(* CODESYS project lateral_levitation_control_new.library
   TcLibraryId: TE140x Module Vendor|lateral_levitation_control_new|0.0.0.4
   Company: TE140x Module Vendor
   Title: lateral_levitation_control_new
   Placeholder: lateral_levitation_control_new
   Version: 0.0.0.4

Project tree, tasks and I/O mapping:
  POUs/
    function block FB_lateral_levitation_control_new [ST]: FB_exit, FB_init, nHResult, eInitExceptionHandling, eUpdateExceptionHandling, nExceptionCnt, stActiveException, bInitialized, bExecute
    TcCOM Wrapper/
      function block FB_lateral_levitation_control_new_TcCOM_InitStruct [ST]: FB_init, FB_afterinit, Reinit, FB_exit, eObjectState, nHResult, ipTcComObject, ipADI, nTaskOid, nTaskPriority, nTaskCycleTimeNs, nTaskPort, nTaskSortOrder, eTraceLevelMax, eModuleCaller, eCallerVerification, eStepSizeAdaptation, eExecutionSequence, bExecute, eAccessLockState, eInitExceptionHandling, eUpdateExceptionHandling, stModuleBuildInfo, bInitialized, nSkippedExecutionCount, stLibraryInfo, stModuleInfo, stModuleGeneratorInfo, stSimulinkModelInfo, elateral_levitation_control_new_P_Sharing, nlateral_levitation_control_new_P_Definer, stlateral_levitation_control_new_P, fSimulationTime, nCycleCount, nExceptionCount, stExceptionInfo
  DUTs/
    data type ST_FB_lateral_levitation_control_new_FB_Main
    data type ST_FB_lateral_levitation_control_new_FB_exit
    data type ST_FB_lateral_levitation_control_new_FB_init
    data type ST_GetSet_HRESULT
    data type E_FpExcptCtrlSetEx
    data type ST_GetSet_E_FpExcptCtrlSetEx
    data type ST_GetSet_ULINT
    data type ST_ExceptionInfo
    data type ST_GetSet_ST_ExceptionInfo
    data type ST_GetSet_BOOL
    data type T_matrix2xdouble
    data type T_matrix4xdouble
    data type E_SimTimeStep
    data type E_SolverMode
    data type E_ssMatrixType
    data type ST_RTWRTModelMethodsInfo
    data type E_slJmBdControl
    data type ST_ssSolverInfo
    data type T_matrix3xdouble
    data type T_matrix4xlogical
    data type ST_B_MATLABFunction2_lateral_levitation_control_new_T
    data type ST_B_lateral_levitation_control_new_T
    data type T_ZCSigState
    data type T_matrix2xZCSigState
    data type ST_PrevZCX_lateral_levitation_control_new_T
    data type ST_X_lateral_levitation_control_new_T
    data type ST_ExtU_lateral_levitation_control_new_T
    data type ST_ExtY_lateral_levitation_control_new_T
    data type T_matrix2xbool
    data type ST_XDis_lateral_levitation_control_new_T
    data type T_matrix8xdouble
    data type T_matrix8x4xdouble
    data type PLREAL
    data type T_matrix4xdoublepointer
    data type ST_ODE4_IntgData
    data type ST_DW_lateral_levitation_control_new_T
    data type ST_x08a7a7bbd0e5d629f7d70ceec84eacfe
    data type ST_xf09845edab6c83520d8d57def6d6fe1c
    data type ST_RT_MODEL_lateral_levitation_control_new_T
    data type T_matrix14xdouble
    data type T_matrix112xdouble
    data type ST_P_lateral_levitation_control_new_T
    data type E_ModuleCaller
    data type E_CallerVerification
    data type E_StepSizeAdaptation
    data type E_ExecutionSequence1
    data type E_FpExcptCtrlSet
    data type ST_TcMatSim_ModuleGeneratorInfo
    data type ST_TcMatSim_SimulinkModelInfo
    data type E_ParameterSharingType
    data type ST_FB_lateral_levitation_control_new_TcCOM_InitStruct
    data type ST_FB_lateral_levitation_control_new_TcCOM_InitStruct_FB_init
    data type ST_FB_lateral_levitation_control_new_TcCOM_InitStruct_FB_afterinit
    data type ST_FB_lateral_levitation_control_new_TcCOM_InitStruct_Reinit
    data type ST_FB_lateral_levitation_control_new_TcCOM_InitStruct_FB_Main
    data type ST_FB_lateral_levitation_control_new_TcCOM_InitStruct_FB_exit
    data type ST_GetSet_TCOM_STATE
    data type ST_GetSet_ITComObject
    data type ST_GetSet_ITcADI
    data type ST_lateral_levitation_control_new_U_T
    data type ST_lateral_levitation_control_new_Y_T
    data type ST_lateral_levitation_control_new_X_T
    data type ST_lateral_levitation_control_new_DW_T
    data type ST_GetSet_OTCID
    data type ST_GetSet_UDINT
    data type ST_GetSet_UINT
    data type ST_GetSet_TcTraceLevel
    data type ST_GetSet_E_ModuleCaller
    data type ST_GetSet_E_CallerVerification
    data type ST_GetSet_E_StepSizeAdaptation
    data type ST_GetSet_E_ExecutionSequence1
    data type ST_GetSet_E_FpExcptCtrlSet
    data type ST_ModuleBuildInfo
    data type ST_GetSet_ST_ModuleBuildInfo
    data type ST_LibraryInfo
    data type ST_GetSet_ST_LibraryInfo
    data type ST_ModuleInfo
    data type ST_GetSet_ST_ModuleInfo
    data type ST_GetSet_ST_TcMatSim_ModuleGeneratorInfo
    data type ST_GetSet_ST_TcMatSim_SimulinkModelInfo
    data type ST_GetSet_E_ParameterSharingType
    data type ST_GetSet_ST_P_lateral_levitation_control_new_T
    data type ST_GetSet_LREAL
  Version/
    global variables Global_Version
*)

// DUTs/ST_FB_lateral_levitation_control_new_FB_Main
{attribute 'TcIecLibraryType'}
{attribute 'hide'}
TYPE ST_FB_lateral_levitation_control_new_FB_Main : 
	STRUCT
		{attribute 'GUID' := '18071995-0000-0000-0000-000000000018'}
		pInst : PVOID;
		result : BOOL;
		 {attribute 'hide'}
		_reserved1 : UINT_24_56;
	END_STRUCT
END_TYPE

// DUTs/ST_FB_lateral_levitation_control_new_FB_exit
{attribute 'TcIecLibraryType'}
{attribute 'hide'}
TYPE ST_FB_lateral_levitation_control_new_FB_exit : 
	STRUCT
		{attribute 'GUID' := '18071995-0000-0000-0000-000000000018'}
		pInst : PVOID;
		bInCopyCode : BOOL;
		result : BOOL;
		 {attribute 'hide'}
		_reserved1 : UINT_16_48;
	END_STRUCT
END_TYPE

// DUTs/ST_FB_lateral_levitation_control_new_FB_init
{attribute 'TcIecLibraryType'}
{attribute 'hide'}
TYPE ST_FB_lateral_levitation_control_new_FB_init : 
	STRUCT
		{attribute 'GUID' := '18071995-0000-0000-0000-000000000018'}
		pInst : PVOID;
		bInitRetains : BOOL;
		bInCopyCode : BOOL;
		result : BOOL;
		 {attribute 'hide'}
		_reserved1 : UINT_8_40;
	END_STRUCT
END_TYPE

// DUTs/ST_GetSet_HRESULT
{attribute 'TcIecLibraryType'}
{attribute 'hide'}
TYPE ST_GetSet_HRESULT : 
	STRUCT
		{attribute 'GUID' := '18071995-0000-0000-0000-000000000018'}
		pInst : PVOID;
		{attribute 'GUID' := '18071995-0000-0000-0000-000000000019'}
		nParam : HRESULT;
		 {attribute 'hide'}
		_reserved1 : UINT_0_32;
	END_STRUCT
END_TYPE

// DUTs/E_FpExcptCtrlSetEx
(* Generated from type 'TcMgSdk.FpExcptCtrlSetEx' *)
{attribute 'TcIecLibraryType'}
TYPE E_FpExcptCtrlSetEx : (
	CallerExceptions:=1, 	(* Use the floating point exception settings provided by the caller *)
	ThrowExceptions:=3, 	(* Enable floating point exceptions on invalid operations and divisions by zero *)
	SuppressExceptions:=13, 	(* Disable floating point exceptions. *)
	LogExceptions:=19, 	(* Log exception information. *)
	LogAndHold:=51, 	(* Log exception information and puase execution of the cyclic code after completion of the actual cycle *)
	LogAndCatch:=83, 	(* Log exception information and immediately terminate execution of the cyclic code. Reinitialization is required to restart. *)
	LogAndDump:=147, 	(* Log exception information, create a dump file with detailed exception information and try to continue execution of the cyclic code *)
	LogHoldAndDump:=179, 	(* Log exception information, create a dump file with detailed exception information and puase execution of the cyclic code after completion of the actual cycle *)
	LogCatchAndDump:=211	(* Log exception information, create a dump file with detailed exception information and immediately terminate execution of the cyclic code. Reinitialization is required to restart. *)
) USINT;
END_TYPE

// DUTs/ST_GetSet_E_FpExcptCtrlSetEx
{attribute 'TcIecLibraryType'}
{attribute 'hide'}
TYPE ST_GetSet_E_FpExcptCtrlSetEx : 
	STRUCT
		{attribute 'GUID' := '18071995-0000-0000-0000-000000000018'}
		pInst : PVOID;
		eParam : E_FpExcptCtrlSetEx;
		 {attribute 'hide'}
		_reserved1 : UINT_24_56;
	END_STRUCT
END_TYPE

// DUTs/ST_GetSet_ULINT
{attribute 'TcIecLibraryType'}
{attribute 'hide'}
TYPE ST_GetSet_ULINT : 
	STRUCT
		{attribute 'GUID' := '18071995-0000-0000-0000-000000000018'}
		pInst : PVOID;
		nParam : ULINT;
	END_STRUCT
END_TYPE

// DUTs/ST_ExceptionInfo
(* Generated from type 'TcMgSdk.ExceptionInfo' *)
{attribute 'TcIecLibraryType'}
TYPE ST_ExceptionInfo : 
	STRUCT
		(* Generated from item 'ExceptionCode' *)
		nExceptionCode : DINT;
		(* Generated from item 'TmxName' *)
		{attribute 'GUID' := '18071995-0000-0000-0000-00010000007F'}
		sTmxName : STRING(127);
		(* Generated from item 'TmxVersion' *)
		nTmxVersion : ARRAY [0..3] OF UDINT;
		(* Generated from item 'InstructionAddr' *)
		nInstructionAddr : UDINT;
		(* Generated from item 'ReturnAddr' *)
		nReturnAddr : ARRAY [0..3] OF UDINT;
		(* Generated from item 'DumpCreated' *)
		bDumpCreated : BOOL;
		 {attribute 'hide'}
		_reserved1 : ARRAY [1..3] OF USINT;
	END_STRUCT
END_TYPE

// DUTs/ST_GetSet_ST_ExceptionInfo
{attribute 'TcIecLibraryType'}
{attribute 'hide'}
TYPE ST_GetSet_ST_ExceptionInfo : 
	STRUCT
		{attribute 'GUID' := '18071995-0000-0000-0000-000000000018'}
		pInst : PVOID;
		stParam : ST_ExceptionInfo;
		 {attribute 'hide'}
		_reserved1 : UINT_0_32;
	END_STRUCT
END_TYPE

// DUTs/ST_GetSet_BOOL
{attribute 'TcIecLibraryType'}
{attribute 'hide'}
TYPE ST_GetSet_BOOL : 
	STRUCT
		{attribute 'GUID' := '18071995-0000-0000-0000-000000000018'}
		pInst : PVOID;
		bParam : BOOL;
		 {attribute 'hide'}
		_reserved1 : UINT_24_56;
	END_STRUCT
END_TYPE

// DUTs/T_matrix2xdouble
(* Generated from type 'matrix2xdouble' *)
{attribute 'TcIecLibraryType'}
TYPE T_matrix2xdouble : ARRAY [0..1] OF LREAL;
END_TYPE

// DUTs/T_matrix4xdouble
(* Generated from type 'matrix4xdouble' *)
{attribute 'TcIecLibraryType'}
TYPE T_matrix4xdouble : ARRAY [0..3] OF LREAL;
END_TYPE

// DUTs/E_SimTimeStep
(* Generated from type 'SimTimeStep' *)
{attribute 'TcIecLibraryType'}
{attribute 'qualified_only' := 'true'}
TYPE E_SimTimeStep : (MINOR_TIME_STEP:=0, MAJOR_TIME_STEP:=1) DINT;
END_TYPE

// DUTs/E_SolverMode
(* Generated from type 'SolverMode' *)
{attribute 'TcIecLibraryType'}
{attribute 'qualified_only' := 'true'}
TYPE E_SolverMode : (SOLVER_MODE_AUTO:=0, SOLVER_MODE_SINGLETASKING:=1, SOLVER_MODE_MULTITASKING:=2) DINT;
END_TYPE

// DUTs/E_ssMatrixType
(* Generated from type 'ssMatrixType' *)
{attribute 'TcIecLibraryType'}
{attribute 'qualified_only' := 'true'}
TYPE E_ssMatrixType : (SS_MATRIX_NONE:=0, SS_MATRIX_CONSTANT:=1, SS_MATRIX_TIMEDEP:=2, SS_MATRIX_STATEDEP:=3) DINT;
END_TYPE

// DUTs/ST_RTWRTModelMethodsInfo
(* Generated from type 'RTWRTModelMethodsInfo' *)
{attribute 'TcIecLibraryType'}
TYPE ST_RTWRTModelMethodsInfo : 
	STRUCT
		(* Generated from item 'rtModelPtr' *)
		{attribute 'GUID' := '18071995-0000-0000-0000-000000000018'}
		prtModelPtr : PVOID;
		(* Generated from item 'rtmInitSizesFcn' *)
		{attribute 'GUID' := '18071995-0000-0000-0000-000000000018'}
		prtmInitSizesFcn : PVOID;
		(* Generated from item 'rtmInitSampTimesFcn' *)
		{attribute 'GUID' := '18071995-0000-0000-0000-000000000018'}
		prtmInitSampTimesFcn : PVOID;
		(* Generated from item 'rtmStartFcn' *)
		{attribute 'GUID' := '18071995-0000-0000-0000-000000000018'}
		prtmStartFcn : PVOID;
		(* Generated from item 'rtmOutputsFcn' *)
		{attribute 'GUID' := '18071995-0000-0000-0000-000000000018'}
		prtmOutputsFcn : PVOID;
		(* Generated from item 'rtmUpdateFcn' *)
		{attribute 'GUID' := '18071995-0000-0000-0000-000000000018'}
		prtmUpdateFcn : PVOID;
		(* Generated from item 'rtmDervisFcn' *)
		{attribute 'GUID' := '18071995-0000-0000-0000-000000000018'}
		prtmDervisFcn : PVOID;
		(* Generated from item 'rtmProjectionFcn' *)
		{attribute 'GUID' := '18071995-0000-0000-0000-000000000018'}
		prtmProjectionFcn : PVOID;
		(* Generated from item 'rtmMassMatrixFcn' *)
		{attribute 'GUID' := '18071995-0000-0000-0000-000000000018'}
		prtmMassMatrixFcn : PVOID;
		(* Generated from item 'rtmForcingFunctionFcn' *)
		{attribute 'GUID' := '18071995-0000-0000-0000-000000000018'}
		prtmForcingFunctionFcn : PVOID;
		(* Generated from item 'rtmTerminateFcn' *)
		{attribute 'GUID' := '18071995-0000-0000-0000-000000000018'}
		prtmTerminateFcn : PVOID;
		(* Generated from item 'rtmDiscreteEventsFcn' *)
		{attribute 'GUID' := '18071995-0000-0000-0000-000000000018'}
		prtmDiscreteEventsFcn : PVOID;
	END_STRUCT
END_TYPE

// DUTs/E_slJmBdControl
(* Generated from type 'slJmBdControl' *)
{attribute 'TcIecLibraryType'}
{attribute 'qualified_only' := 'true'}
TYPE E_slJmBdControl : (SL_JM_BD_AUTO:=0, SL_JM_BD_SPARSE_PERTURBATION:=1, SL_JM_BD_FULL_PERTURBATION:=2, SL_JM_BD_SPARSE_ANALYTICAL:=3, SL_JM_BD_FULL_ANALYTICAL:=4) DINT;
END_TYPE

// DUTs/ST_ssSolverInfo
(* Generated from type 'ssSolverInfo' *)
{attribute 'TcIecLibraryType'}
TYPE ST_ssSolverInfo : 
	STRUCT
		(* Generated from item 'rtModelPtr' *)
		{attribute 'GUID' := '18071995-0000-0000-0000-000000000018'}
		prtModelPtr : PVOID;
		simTimeStepPtr : POINTER TO E_SimTimeStep;
		(* Generated from item 'solverData' *)
		{attribute 'GUID' := '18071995-0000-0000-0000-000000000018'}
		psolverData : PVOID;
		solverName : POINTER TO SINT;
		(* Generated from item 'isVariableStepSolver' *)
		bisVariableStepSolver : BOOL;
		(* Generated from item 'solverNeedsReset' *)
		bsolverNeedsReset : BOOL;
		 {attribute 'hide'}
		_reserved1 : UINT;
		(* Generated from item 'solverMode' *)
		esolverMode : E_SolverMode;
		(* Generated from item 'solverStopTime' *)
		fsolverStopTime : LREAL;
		stepSizePtr : POINTER TO LREAL;
		(* Generated from item 'minStepSize' *)
		fminStepSize : LREAL;
		(* Generated from item 'maxStepSize' *)
		fmaxStepSize : LREAL;
		(* Generated from item 'fixedStepSize' *)
		ffixedStepSize : LREAL;
		(* Generated from item 'solverShapePreserveControl' *)
		nsolverShapePreserveControl : DINT;
		(* Generated from item 'solverMaxConsecutiveMinStep' *)
		nsolverMaxConsecutiveMinStep : DINT;
		(* Generated from item 'maxNumMinSteps' *)
		nmaxNumMinSteps : DINT;
		(* Generated from item 'solverMaxOrder' *)
		nsolverMaxOrder : DINT;
		(* Generated from item 'solverConsecutiveZCsStepRelTol' *)
		fsolverConsecutiveZCsStepRelTol : LREAL;
		(* Generated from item 'solverMaxConsecutiveZCs' *)
		nsolverMaxConsecutiveZCs : DINT;
		(* Generated from item 'solverExtrapolationOrder' *)
		nsolverExtrapolationOrder : DINT;
		(* Generated from item 'solverNumberNewtonIterations' *)
		nsolverNumberNewtonIterations : DINT;
		(* Generated from item 'solverRefineFactor' *)
		nsolverRefineFactor : DINT;
		(* Generated from item 'solverRelTol' *)
		fsolverRelTol : LREAL;
		(* Generated from item 'unused_real_T_1' *)
		funused_real_T_1 : LREAL;
		dXPtr : POINTER TO POINTER TO LREAL;
		tPtr : POINTER TO POINTER TO LREAL;
		numContStatesPtr : POINTER TO DINT;
		contStatesPtr : POINTER TO POINTER TO LREAL;
		numPeriodicContStatesPtr : POINTER TO DINT;
		periodicContStateIndicesPtr : POINTER TO POINTER TO DINT;
		periodicContStateRangesPtr : POINTER TO POINTER TO LREAL;
		zcSignalVector : POINTER TO LREAL;
		zcEventsVector : POINTER TO USINT;
		zcSignalAttrib : POINTER TO USINT;
		(* Generated from item 'zcSignalVectorLength' *)
		nzcSignalVectorLength : DINT;
		 {attribute 'hide'}
		_reserved2 : UINT_0_32;
		reserved : POINTER TO USINT;
		(* Generated from item 'foundContZcEvents' *)
		bfoundContZcEvents : BOOL;
		(* Generated from item 'isAtLeftPostOfContZcEvent' *)
		bisAtLeftPostOfContZcEvent : BOOL;
		(* Generated from item 'isAtRightPostOfContZcEvent' *)
		bisAtRightPostOfContZcEvent : BOOL;
		(* Generated from item 'adaptiveZcDetection' *)
		badaptiveZcDetection : BOOL;
		(* Generated from item 'numZcSignals' *)
		nnumZcSignals : DINT;
		(* Generated from item 'stateProjection' *)
		bstateProjection : BOOL;
		(* Generated from item 'robustResetMethod' *)
		brobustResetMethod : BOOL;
		(* Generated from item 'updateJacobianAtReset' *)
		bupdateJacobianAtReset : BOOL;
		(* Generated from item 'consistencyChecking' *)
		bconsistencyChecking : BOOL;
		(* Generated from item 'massMatrixType' *)
		emassMatrixType : E_ssMatrixType;
		(* Generated from item 'massMatrixNzMax' *)
		nmassMatrixNzMax : DINT;
		 {attribute 'hide'}
		_reserved3 : UINT_0_32;
		massMatrixIr : POINTER TO DINT;
		massMatrixJc : POINTER TO DINT;
		massMatrixPr : POINTER TO LREAL;
		errStatusPtr : POINTER TO POINTER TO SINT;
		modelMethodsPtr : POINTER TO ST_RTWRTModelMethodsInfo;
		(* Generated from item 'zcThreshold' *)
		fzcThreshold : LREAL;
		(* Generated from item 'reserved_1' *)
		nreserved_1 : DINT;
		(* Generated from item 'consecutiveZCsError' *)
		nconsecutiveZCsError : DINT;
		(* Generated from item 'CTOutputIncnstWithState' *)
		bCTOutputIncnstWithState : BOOL;
		(* Generated from item 'isComputingJacobian' *)
		bisComputingJacobian : BOOL;
		 {attribute 'hide'}
		_reserved4 : UINT;
		(* Generated from item 'solverJacobianMethodControl' *)
		esolverJacobianMethodControl : E_slJmBdControl;
		(* Generated from item 'ignoredZcDiagnostic' *)
		nignoredZcDiagnostic : DINT;
		(* Generated from item 'maskedZcDiagnostic' *)
		nmaskedZcDiagnostic : DINT;
		(* Generated from item 'isOutputMethodComputed' *)
		bisOutputMethodComputed : BOOL;
		 {attribute 'hide'}
		_reserved5 : ARRAY [1..3] OF USINT;
		(* Generated from item 'maxZcBracketingIterations' *)
		nmaxZcBracketingIterations : DINT;
		(* Generated from item 'isMinorTimeStepWithModeChange' *)
		bisMinorTimeStepWithModeChange : BOOL;
		 {attribute 'hide'}
		_reserved6 : ARRAY [1..3] OF USINT;
		(* Generated from item 'maxZcPerStep' *)
		nmaxZcPerStep : DINT;
		zcSignalPtr : POINTER TO POINTER TO LREAL;
		(* Generated from item 'contStateDisabledPtr' *)
		bcontStateDisabledPtr : POINTER TO POINTER TO BOOL;
		(* Generated from item 'isContModeFrozen' *)
		bisContModeFrozen : BOOL;
		 {attribute 'hide'}
		_reserved7 : ARRAY [1..7] OF USINT;
	END_STRUCT
END_TYPE

// DUTs/T_matrix3xdouble
(* Generated from type 'matrix3xdouble' *)
{attribute 'TcIecLibraryType'}
TYPE T_matrix3xdouble : ARRAY [0..2] OF LREAL;
END_TYPE

// DUTs/T_matrix4xlogical
(* Generated from type 'matrix4xlogical' *)
{attribute 'TcIecLibraryType'}
{attribute 'BaseTypeGUID' := '18071995-0000-0000-0000-000000000030'}
TYPE T_matrix4xlogical : ARRAY [0..3] OF BOOL;
END_TYPE

// DUTs/ST_B_MATLABFunction2_lateral_levitation_control_new_T
(* Generated from type 'B_MATLABFunction2_lateral_levitation_control_new_T' *)
{attribute 'TcIecLibraryType'}
TYPE ST_B_MATLABFunction2_lateral_levitation_control_new_T : 
	STRUCT
		(* Generated from item 'y' *)
		ay : T_matrix4xdouble;
	END_STRUCT
END_TYPE

// DUTs/ST_B_lateral_levitation_control_new_T
(* Generated from type 'B_lateral_levitation_control_new_T' *)
{attribute 'TcIecLibraryType'}
TYPE ST_B_lateral_levitation_control_new_T : 
	STRUCT
		(* Generated from item 'levi_operational_y_PID' *)
		flevi_operational_y_PID : LREAL;
		(* Generated from item 'K_F_y' *)
		fK_F_y : LREAL;
		(* Generated from item 'levi_operational_yaw_PID' *)
		flevi_operational_yaw_PID : LREAL;
		(* Generated from item 'K_F_yaw' *)
		fK_F_yaw : LREAL;
		(* Generated from item 'UnitDelay' *)
		aUnitDelay : T_matrix2xdouble;
		(* Generated from item 'Switch1' *)
		aSwitch1 : T_matrix2xdouble;
		(* Generated from item 'Switch3' *)
		aSwitch3 : T_matrix2xdouble;
		(* Generated from item 'Add4' *)
		fAdd4 : LREAL;
		(* Generated from item 'UnitDelay1' *)
		fUnitDelay1 : LREAL;
		(* Generated from item 'Add4_c' *)
		fAdd4_c : LREAL;
		(* Generated from item 'UnitDelay1_d' *)
		fUnitDelay1_d : LREAL;
		(* Generated from item 'Add4_cu' *)
		fAdd4_cu : LREAL;
		(* Generated from item 'UnitDelay1_o' *)
		fUnitDelay1_o : LREAL;
		(* Generated from item 'Add4_d' *)
		fAdd4_d : LREAL;
		(* Generated from item 'UnitDelay1_j' *)
		fUnitDelay1_j : LREAL;
		(* Generated from item 'Add4_k' *)
		fAdd4_k : LREAL;
		(* Generated from item 'UnitDelay1_f' *)
		fUnitDelay1_f : LREAL;
		(* Generated from item 'Add4_l' *)
		fAdd4_l : LREAL;
		(* Generated from item 'UnitDelay1_c' *)
		fUnitDelay1_c : LREAL;
		(* Generated from item 'Add4_d1' *)
		fAdd4_d1 : LREAL;
		(* Generated from item 'UnitDelay1_m' *)
		fUnitDelay1_m : LREAL;
		(* Generated from item 'Switch1_a' *)
		fSwitch1_a : LREAL;
		(* Generated from item 'Add4_o' *)
		fAdd4_o : LREAL;
		(* Generated from item 'UnitDelay1_k' *)
		fUnitDelay1_k : LREAL;
		(* Generated from item 'Add4_l5' *)
		fAdd4_l5 : LREAL;
		(* Generated from item 'UnitDelay1_c3' *)
		fUnitDelay1_c3 : LREAL;
		(* Generated from item 'Add4_g' *)
		fAdd4_g : LREAL;
		(* Generated from item 'UnitDelay1_b' *)
		fUnitDelay1_b : LREAL;
		(* Generated from item 'Add4_o4' *)
		fAdd4_o4 : LREAL;
		(* Generated from item 'UnitDelay1_mq' *)
		fUnitDelay1_mq : LREAL;
		(* Generated from item 'Add4_dn' *)
		fAdd4_dn : LREAL;
		(* Generated from item 'UnitDelay1_b0' *)
		fUnitDelay1_b0 : LREAL;
		(* Generated from item 'Add4_p' *)
		fAdd4_p : LREAL;
		(* Generated from item 'UnitDelay1_fa' *)
		fUnitDelay1_fa : LREAL;
		(* Generated from item 'Add4_j' *)
		fAdd4_j : LREAL;
		(* Generated from item 'UnitDelay1_b0w' *)
		fUnitDelay1_b0w : LREAL;
		(* Generated from item 'Switch1_c' *)
		fSwitch1_c : LREAL;
		(* Generated from item 'Sum4' *)
		aSum4 : T_matrix2xdouble;
		(* Generated from item 'Switch4' *)
		aSwitch4 : T_matrix2xdouble;
		(* Generated from item 'Switch2' *)
		aSwitch2 : T_matrix4xdouble;
		(* Generated from item 'Add5' *)
		fAdd5 : LREAL;
		(* Generated from item 'Add6' *)
		fAdd6 : LREAL;
		(* Generated from item 'Gain' *)
		fGain : LREAL;
		(* Generated from item 'UnitDelay2' *)
		fUnitDelay2 : LREAL;
		(* Generated from item 'Sum4_p' *)
		fSum4_p : LREAL;
		(* Generated from item 'Sum5' *)
		fSum5 : LREAL;
		(* Generated from item 'Add5_g' *)
		fAdd5_g : LREAL;
		(* Generated from item 'Add6_g' *)
		fAdd6_g : LREAL;
		(* Generated from item 'Gain_b' *)
		fGain_b : LREAL;
		(* Generated from item 'UnitDelay2_b' *)
		fUnitDelay2_b : LREAL;
		(* Generated from item 'Sum4_f' *)
		fSum4_f : LREAL;
		(* Generated from item 'Sum5_j' *)
		fSum5_j : LREAL;
		(* Generated from item 'Add5_k' *)
		fAdd5_k : LREAL;
		(* Generated from item 'Add6_i' *)
		fAdd6_i : LREAL;
		(* Generated from item 'Gain_e' *)
		fGain_e : LREAL;
		(* Generated from item 'UnitDelay2_h' *)
		fUnitDelay2_h : LREAL;
		(* Generated from item 'Sum4_i' *)
		fSum4_i : LREAL;
		(* Generated from item 'Sum5_p' *)
		fSum5_p : LREAL;
		(* Generated from item 'Add5_c' *)
		fAdd5_c : LREAL;
		(* Generated from item 'Add6_a' *)
		fAdd6_a : LREAL;
		(* Generated from item 'Gain_l' *)
		fGain_l : LREAL;
		(* Generated from item 'UnitDelay2_i' *)
		fUnitDelay2_i : LREAL;
		(* Generated from item 'Sum4_pp' *)
		fSum4_pp : LREAL;
		(* Generated from item 'Sum5_l' *)
		fSum5_l : LREAL;
		(* Generated from item 'Add5_d' *)
		fAdd5_d : LREAL;
		(* Generated from item 'Add6_m' *)
		fAdd6_m : LREAL;
		(* Generated from item 'Gain_n' *)
		fGain_n : LREAL;
		(* Generated from item 'UnitDelay2_o' *)
		fUnitDelay2_o : LREAL;
		(* Generated from item 'Sum4_b' *)
		fSum4_b : LREAL;
		(* Generated from item 'Sum5_n' *)
		fSum5_n : LREAL;
		(* Generated from item 'Add5_a' *)
		fAdd5_a : LREAL;
		(* Generated from item 'Add6_d' *)
		fAdd6_d : LREAL;
		(* Generated from item 'Gain_j' *)
		fGain_j : LREAL;
		(* Generated from item 'UnitDelay2_ot' *)
		fUnitDelay2_ot : LREAL;
		(* Generated from item 'Sum4_j' *)
		fSum4_j : LREAL;
		(* Generated from item 'Sum5_l0' *)
		fSum5_l0 : LREAL;
		(* Generated from item 'Add5_e' *)
		fAdd5_e : LREAL;
		(* Generated from item 'Add6_o' *)
		fAdd6_o : LREAL;
		(* Generated from item 'Gain_i' *)
		fGain_i : LREAL;
		(* Generated from item 'UnitDelay2_c' *)
		fUnitDelay2_c : LREAL;
		(* Generated from item 'Sum4_ia' *)
		fSum4_ia : LREAL;
		(* Generated from item 'Sum5_i' *)
		fSum5_i : LREAL;
		(* Generated from item 'Add5_f' *)
		fAdd5_f : LREAL;
		(* Generated from item 'Add6_f' *)
		fAdd6_f : LREAL;
		(* Generated from item 'Gain_k' *)
		fGain_k : LREAL;
		(* Generated from item 'UnitDelay2_n' *)
		fUnitDelay2_n : LREAL;
		(* Generated from item 'Sum4_b4' *)
		fSum4_b4 : LREAL;
		(* Generated from item 'Sum5_c' *)
		fSum5_c : LREAL;
		(* Generated from item 'Add5_p' *)
		fAdd5_p : LREAL;
		(* Generated from item 'Add6_b' *)
		fAdd6_b : LREAL;
		(* Generated from item 'Gain_g' *)
		fGain_g : LREAL;
		(* Generated from item 'UnitDelay2_ni' *)
		fUnitDelay2_ni : LREAL;
		(* Generated from item 'Sum4_l' *)
		fSum4_l : LREAL;
		(* Generated from item 'Sum5_j1' *)
		fSum5_j1 : LREAL;
		(* Generated from item 'Add5_o' *)
		fAdd5_o : LREAL;
		(* Generated from item 'Add6_k' *)
		fAdd6_k : LREAL;
		(* Generated from item 'Gain_a' *)
		fGain_a : LREAL;
		(* Generated from item 'UnitDelay2_h2' *)
		fUnitDelay2_h2 : LREAL;
		(* Generated from item 'Sum4_ir' *)
		fSum4_ir : LREAL;
		(* Generated from item 'Sum5_pd' *)
		fSum5_pd : LREAL;
		(* Generated from item 'Add5_l' *)
		fAdd5_l : LREAL;
		(* Generated from item 'Add6_bx' *)
		fAdd6_bx : LREAL;
		(* Generated from item 'Gain_gq' *)
		fGain_gq : LREAL;
		(* Generated from item 'UnitDelay2_bx' *)
		fUnitDelay2_bx : LREAL;
		(* Generated from item 'Sum4_ph' *)
		fSum4_ph : LREAL;
		(* Generated from item 'Sum5_ni' *)
		fSum5_ni : LREAL;
		(* Generated from item 'Add5_cz' *)
		fAdd5_cz : LREAL;
		(* Generated from item 'Add6_e' *)
		fAdd6_e : LREAL;
		(* Generated from item 'Gain_im' *)
		fGain_im : LREAL;
		(* Generated from item 'UnitDelay2_p' *)
		fUnitDelay2_p : LREAL;
		(* Generated from item 'Sum4_c' *)
		fSum4_c : LREAL;
		(* Generated from item 'Sum5_m' *)
		fSum5_m : LREAL;
		(* Generated from item 'Add5_i' *)
		fAdd5_i : LREAL;
		(* Generated from item 'Add6_p' *)
		fAdd6_p : LREAL;
		(* Generated from item 'Gain_nv' *)
		fGain_nv : LREAL;
		(* Generated from item 'UnitDelay2_ct' *)
		fUnitDelay2_ct : LREAL;
		(* Generated from item 'Sum4_l0' *)
		fSum4_l0 : LREAL;
		(* Generated from item 'Sum5_jx' *)
		fSum5_jx : LREAL;
		(* Generated from item 'Add5_m' *)
		fAdd5_m : LREAL;
		(* Generated from item 'Add6_pa' *)
		fAdd6_pa : LREAL;
		(* Generated from item 'Gain_k5' *)
		fGain_k5 : LREAL;
		(* Generated from item 'UnitDelay2_e' *)
		fUnitDelay2_e : LREAL;
		(* Generated from item 'Sum4_e' *)
		fSum4_e : LREAL;
		(* Generated from item 'Sum5_g' *)
		fSum5_g : LREAL;
		(* Generated from item 'IsPeak1' *)
		aIsPeak1 : T_matrix2xdouble;
		(* Generated from item 'Switch2_e' *)
		aSwitch2_e : T_matrix2xdouble;
		(* Generated from item 'Sum' *)
		fSum : LREAL;
		(* Generated from item 'Sum1' *)
		fSum1 : LREAL;
		(* Generated from item 'clamptot' *)
		fclamptot : LREAL;
		(* Generated from item 'Sum_b' *)
		fSum_b : LREAL;
		(* Generated from item 'Sum1_h' *)
		fSum1_h : LREAL;
		(* Generated from item 'clamptot_e' *)
		fclamptot_e : LREAL;
		(* Generated from item 'K_I_yaw' *)
		fK_I_yaw : LREAL;
		(* Generated from item 'K_I_y' *)
		fK_I_y : LREAL;
		(* Generated from item 'current_reqf' *)
		fcurrent_reqf : LREAL;
		(* Generated from item 'current_reqb' *)
		fcurrent_reqb : LREAL;
		(* Generated from item 'current_reqf_e' *)
		fcurrent_reqf_e : LREAL;
		(* Generated from item 'current_reqb_o' *)
		fcurrent_reqb_o : LREAL;
		(* Generated from item 'Is' *)
		aIs : T_matrix2xdouble;
		(* Generated from item 'satmin' *)
		asatmin : T_matrix2xdouble;
		(* Generated from item 'satmax' *)
		asatmax : T_matrix2xdouble;
		(* Generated from item 'displ_fb' *)
		adispl_fb : T_matrix2xdouble;
		(* Generated from item 'airgap_diff' *)
		fairgap_diff : LREAL;
		(* Generated from item 'Fy' *)
		fFy : LREAL;
		(* Generated from item 'tau_z' *)
		ftau_z : LREAL;
		(* Generated from item 'F_ems' *)
		aF_ems : T_matrix2xdouble;
		(* Generated from item 'clamp_y' *)
		aclamp_y : T_matrix2xdouble;
		(* Generated from item 'clamp_psi' *)
		aclamp_psi : T_matrix2xdouble;
		(* Generated from item 'counter' *)
		acounter : T_matrix3xdouble;
		(* Generated from item 'q' *)
		fq : LREAL;
		(* Generated from item 'q_f' *)
		fq_f : LREAL;
		(* Generated from item 'q_h' *)
		fq_h : LREAL;
		(* Generated from item 'q_n' *)
		fq_n : LREAL;
		(* Generated from item 'q_c' *)
		fq_c : LREAL;
		(* Generated from item 'q_m' *)
		fq_m : LREAL;
		(* Generated from item 'q_p' *)
		fq_p : LREAL;
		(* Generated from item 'q_i' *)
		fq_i : LREAL;
		(* Generated from item 'q_ce' *)
		fq_ce : LREAL;
		(* Generated from item 'q_mb' *)
		fq_mb : LREAL;
		(* Generated from item 'q_l' *)
		fq_l : LREAL;
		(* Generated from item 'q_na' *)
		fq_na : LREAL;
		(* Generated from item 'q_e' *)
		fq_e : LREAL;
		(* Generated from item 'q_g' *)
		fq_g : LREAL;
		(* Generated from item 'UnaryMinus' *)
		fUnaryMinus : LREAL;
		(* Generated from item 'UnaryMinus_o' *)
		fUnaryMinus_o : LREAL;
		(* Generated from item 'UnaryMinus_k' *)
		fUnaryMinus_k : LREAL;
		(* Generated from item 'UnaryMinus_c' *)
		fUnaryMinus_c : LREAL;
		(* Generated from item 'UnaryMinus_m' *)
		fUnaryMinus_m : LREAL;
		(* Generated from item 'UnaryMinus_a' *)
		fUnaryMinus_a : LREAL;
		(* Generated from item 'UnaryMinus_oh' *)
		fUnaryMinus_oh : LREAL;
		(* Generated from item 'UnaryMinus_e' *)
		fUnaryMinus_e : LREAL;
		(* Generated from item 'UnaryMinus_ah' *)
		fUnaryMinus_ah : LREAL;
		(* Generated from item 'UnaryMinus_g' *)
		fUnaryMinus_g : LREAL;
		(* Generated from item 'UnaryMinus_o2' *)
		fUnaryMinus_o2 : LREAL;
		(* Generated from item 'UnaryMinus_n' *)
		fUnaryMinus_n : LREAL;
		(* Generated from item 'UnaryMinus_l' *)
		fUnaryMinus_l : LREAL;
		(* Generated from item 'UnaryMinus_o5' *)
		fUnaryMinus_o5 : LREAL;
		(* Generated from item 't' *)
		ft : LREAL;
		(* Generated from item 's' *)
		fs : LREAL;
		(* Generated from item 'v' *)
		fv : LREAL;
		(* Generated from item 't_j' *)
		ft_j : LREAL;
		(* Generated from item 's_c' *)
		fs_c : LREAL;
		(* Generated from item 'v_h' *)
		fv_h : LREAL;
		(* Generated from item 'Product4' *)
		fProduct4 : LREAL;
		(* Generated from item 't_f' *)
		ft_f : LREAL;
		(* Generated from item 's_k' *)
		fs_k : LREAL;
		(* Generated from item 'v_hr' *)
		fv_hr : LREAL;
		(* Generated from item 'Product4_d' *)
		fProduct4_d : LREAL;
		(* Generated from item 't_i' *)
		ft_i : LREAL;
		(* Generated from item 's_b' *)
		fs_b : LREAL;
		(* Generated from item 'v_a' *)
		fv_a : LREAL;
		(* Generated from item 'Product4_g' *)
		fProduct4_g : LREAL;
		(* Generated from item 't_h' *)
		ft_h : LREAL;
		(* Generated from item 's_n' *)
		fs_n : LREAL;
		(* Generated from item 'Product4_c' *)
		fProduct4_c : LREAL;
		(* Generated from item 't_c' *)
		ft_c : LREAL;
		(* Generated from item 's_e' *)
		fs_e : LREAL;
		(* Generated from item 'Product4_m' *)
		fProduct4_m : LREAL;
		(* Generated from item 't_fb' *)
		ft_fb : LREAL;
		(* Generated from item 's_ke' *)
		fs_ke : LREAL;
		(* Generated from item 't_e' *)
		ft_e : LREAL;
		(* Generated from item 's_i' *)
		fs_i : LREAL;
		(* Generated from item 'v_c' *)
		fv_c : LREAL;
		(* Generated from item 'Product4_b' *)
		fProduct4_b : LREAL;
		(* Generated from item 't_o' *)
		ft_o : LREAL;
		(* Generated from item 's_cr' *)
		fs_cr : LREAL;
		(* Generated from item 'v_n' *)
		fv_n : LREAL;
		(* Generated from item 'Product4_n' *)
		fProduct4_n : LREAL;
		(* Generated from item 't_l' *)
		ft_l : LREAL;
		(* Generated from item 's_ci' *)
		fs_ci : LREAL;
		(* Generated from item 'v_m' *)
		fv_m : LREAL;
		(* Generated from item 'Product4_gh' *)
		fProduct4_gh : LREAL;
		(* Generated from item 't_a' *)
		ft_a : LREAL;
		(* Generated from item 's_h' *)
		fs_h : LREAL;
		(* Generated from item 'v_j' *)
		fv_j : LREAL;
		(* Generated from item 'Product4_k' *)
		fProduct4_k : LREAL;
		(* Generated from item 't_b' *)
		ft_b : LREAL;
		(* Generated from item 's_ne' *)
		fs_ne : LREAL;
		(* Generated from item 'v_d' *)
		fv_d : LREAL;
		(* Generated from item 'Product4_o' *)
		fProduct4_o : LREAL;
		(* Generated from item 't_ip' *)
		ft_ip : LREAL;
		(* Generated from item 's_a' *)
		fs_a : LREAL;
		(* Generated from item 'v_e' *)
		fv_e : LREAL;
		(* Generated from item 't_io' *)
		ft_io : LREAL;
		(* Generated from item 's_ha' *)
		fs_ha : LREAL;
		(* Generated from item 'Abs1' *)
		aAbs1 : T_matrix2xdouble;
		(* Generated from item 'u' *)
		fu : LREAL;
		(* Generated from item 'u_h' *)
		fu_h : LREAL;
		(* Generated from item 'u_f' *)
		fu_f : LREAL;
		(* Generated from item 'u_j' *)
		fu_j : LREAL;
		(* Generated from item 'u_i' *)
		fu_i : LREAL;
		(* Generated from item 'u_m' *)
		fu_m : LREAL;
		(* Generated from item 'u_hh' *)
		fu_hh : LREAL;
		(* Generated from item 'u_n' *)
		fu_n : LREAL;
		(* Generated from item 'u_e' *)
		fu_e : LREAL;
		(* Generated from item 'u_mx' *)
		fu_mx : LREAL;
		(* Generated from item 'u_d' *)
		fu_d : LREAL;
		(* Generated from item 'u_mi' *)
		fu_mi : LREAL;
		(* Generated from item 'u_mt' *)
		fu_mt : LREAL;
		(* Generated from item 'u_k' *)
		fu_k : LREAL;
		(* Generated from item 'MatrixConcatenate' *)
		aMatrixConcatenate : T_matrix4xdouble;
		(* Generated from item 'Product4_e' *)
		fProduct4_e : LREAL;
		(* Generated from item 'Product3' *)
		fProduct3 : LREAL;
		(* Generated from item 'Product3_o' *)
		fProduct3_o : LREAL;
		(* Generated from item 'Product4_cl' *)
		fProduct4_cl : LREAL;
		(* Generated from item 'Product4_ey' *)
		fProduct4_ey : LREAL;
		(* Generated from item 'Product4_i' *)
		fProduct4_i : LREAL;
		(* Generated from item 'Product3_k' *)
		fProduct3_k : LREAL;
		(* Generated from item 'Product3_c' *)
		fProduct3_c : LREAL;
		(* Generated from item 'Product3_f' *)
		fProduct3_f : LREAL;
		(* Generated from item 'Product3_ov' *)
		fProduct3_ov : LREAL;
		(* Generated from item 'Product3_d' *)
		fProduct3_d : LREAL;
		(* Generated from item 'Product3_f2' *)
		fProduct3_f2 : LREAL;
		(* Generated from item 'Sign' *)
		fSign : LREAL;
		(* Generated from item 'Product4_mn' *)
		fProduct4_mn : LREAL;
		(* Generated from item 'Integrator' *)
		fIntegrator : LREAL;
		(* Generated from item 'Product1' *)
		fProduct1 : LREAL;
		(* Generated from item 'Product3_a' *)
		fProduct3_a : LREAL;
		(* Generated from item 'Product1_h' *)
		fProduct1_h : LREAL;
		(* Generated from item 'Product1_g' *)
		fProduct1_g : LREAL;
		(* Generated from item 'Product1_k' *)
		fProduct1_k : LREAL;
		(* Generated from item 'Product4_h' *)
		fProduct4_h : LREAL;
		(* Generated from item 'Integrator2' *)
		aIntegrator2 : T_matrix2xdouble;
		(* Generated from item 'Product3_h' *)
		fProduct3_h : LREAL;
		(* Generated from item 'Sign1' *)
		fSign1 : LREAL;
		(* Generated from item 'Product4_ke' *)
		fProduct4_ke : LREAL;
		(* Generated from item 'LowerRelop1' *)
		aLowerRelop1 : T_matrix4xlogical;
		(* Generated from item 'UpperRelop' *)
		aUpperRelop : T_matrix4xlogical;
		(* Generated from item 'RelationalOperator1' *)
		bRelationalOperator1 : BOOL;
		(* Generated from item 'LogicalOperator' *)
		bLogicalOperator : BOOL;
		(* Generated from item 'LogicalOperator1' *)
		bLogicalOperator1 : BOOL;
		 {attribute 'hide'}
		_reserved1 : ARRAY [1..5] OF USINT;
		(* Generated from item 'sf_MATLABFunction3' *)
		stsf_MATLABFunction3 : ST_B_MATLABFunction2_lateral_levitation_control_new_T;
		(* Generated from item 'sf_MATLABFunction2' *)
		stsf_MATLABFunction2 : ST_B_MATLABFunction2_lateral_levitation_control_new_T;
	END_STRUCT
END_TYPE

// DUTs/T_ZCSigState
(* Generated from type 'ZCSigState' *)
{attribute 'TcIecLibraryType'}
TYPE T_ZCSigState : USINT;
END_TYPE

// DUTs/T_matrix2xZCSigState
(* Generated from type 'matrix2xZCSigState' *)
{attribute 'TcIecLibraryType'}
{attribute 'BaseTypeGUID' := 'CF0EC509-8CFA-173E-6D32-2A6837BC8565'}
TYPE T_matrix2xZCSigState : ARRAY [0..1] OF T_ZCSigState;
END_TYPE

// DUTs/ST_PrevZCX_lateral_levitation_control_new_T
(* Generated from type 'PrevZCX_lateral_levitation_control_new_T' *)
{attribute 'TcIecLibraryType'}
TYPE ST_PrevZCX_lateral_levitation_control_new_T : 
	STRUCT
		(* Generated from item 'Integrator_Reset_ZCE' *)
		nIntegrator_Reset_ZCE : T_ZCSigState;
		(* Generated from item 'Integrator_Reset_ZCE_p' *)
		nIntegrator_Reset_ZCE_p : T_ZCSigState;
		(* Generated from item 'Integrator1_Reset_ZCE' *)
		aIntegrator1_Reset_ZCE : T_matrix2xZCSigState;
		(* Generated from item 'Integrator2_Reset_ZCE' *)
		aIntegrator2_Reset_ZCE : T_matrix2xZCSigState;
	END_STRUCT
END_TYPE

// DUTs/ST_X_lateral_levitation_control_new_T
(* Generated from type 'X_lateral_levitation_control_new_T' *)
{attribute 'TcIecLibraryType'}
TYPE ST_X_lateral_levitation_control_new_T : 
	STRUCT
		(* Generated from item 'Integrator_CSTATE' *)
		fIntegrator_CSTATE : LREAL;
		(* Generated from item 'Filtertot_CSTATE' *)
		fFiltertot_CSTATE : LREAL;
		(* Generated from item 'Integrator_CSTATE_d' *)
		fIntegrator_CSTATE_d : LREAL;
		(* Generated from item 'Filtertot_CSTATE_p' *)
		fFiltertot_CSTATE_p : LREAL;
		(* Generated from item 'Integrator1_CSTATE' *)
		aIntegrator1_CSTATE : T_matrix2xdouble;
		(* Generated from item 'Integrator2_CSTATE' *)
		aIntegrator2_CSTATE : T_matrix2xdouble;
	END_STRUCT
END_TYPE

// DUTs/ST_ExtU_lateral_levitation_control_new_T
(* Generated from type 'ExtU_lateral_levitation_control_new_T' *)
{attribute 'TcIecLibraryType'}
TYPE ST_ExtU_lateral_levitation_control_new_T : 
	STRUCT
		(* Generated from item 'y' *)
		fy : LREAL;
		(* Generated from item 'yaw' *)
		fyaw : LREAL;
		(* Generated from item 'motor_Fx_l' *)
		fmotor_Fx_l : LREAL;
		(* Generated from item 'motor_Fx_r' *)
		fmotor_Fx_r : LREAL;
		(* Generated from item 'motor_Fy_l' *)
		fmotor_Fy_l : LREAL;
		(* Generated from item 'motor_Fy_r' *)
		fmotor_Fy_r : LREAL;
		(* Generated from item 'z' *)
		fz : LREAL;
	END_STRUCT
END_TYPE

// DUTs/ST_ExtY_lateral_levitation_control_new_T
(* Generated from type 'ExtY_lateral_levitation_control_new_T' *)
{attribute 'TcIecLibraryType'}
TYPE ST_ExtY_lateral_levitation_control_new_T : 
	STRUCT
		(* Generated from item 'F_latreq' *)
		aF_latreq : T_matrix2xdouble;
		(* Generated from item 'I_ems' *)
		aI_ems : T_matrix4xdouble;
		(* Generated from item 'F_emsfb' *)
		aF_emsfb : T_matrix2xdouble;
		(* Generated from item 'airgaps' *)
		aairgaps : T_matrix4xdouble;
		(* Generated from item 'integrals' *)
		aintegrals : T_matrix2xdouble;
		(* Generated from item 't_peak' *)
		at_peak : T_matrix2xdouble;
		(* Generated from item 'tau_x_ems' *)
		ftau_x_ems : LREAL;
	END_STRUCT
END_TYPE

// DUTs/T_matrix2xbool
(* Generated from type 'matrix2xbool' *)
{attribute 'TcIecLibraryType'}
{attribute 'BaseTypeGUID' := '18071995-0000-0000-0000-000000000030'}
TYPE T_matrix2xbool : ARRAY [0..1] OF BOOL;
END_TYPE

// DUTs/ST_XDis_lateral_levitation_control_new_T
(* Generated from type 'XDis_lateral_levitation_control_new_T' *)
{attribute 'TcIecLibraryType'}
TYPE ST_XDis_lateral_levitation_control_new_T : 
	STRUCT
		(* Generated from item 'Integrator_CSTATE' *)
		bIntegrator_CSTATE : BOOL;
		(* Generated from item 'Filtertot_CSTATE' *)
		bFiltertot_CSTATE : BOOL;
		(* Generated from item 'Integrator_CSTATE_d' *)
		bIntegrator_CSTATE_d : BOOL;
		(* Generated from item 'Filtertot_CSTATE_p' *)
		bFiltertot_CSTATE_p : BOOL;
		(* Generated from item 'Integrator1_CSTATE' *)
		aIntegrator1_CSTATE : T_matrix2xbool;
		(* Generated from item 'Integrator2_CSTATE' *)
		aIntegrator2_CSTATE : T_matrix2xbool;
	END_STRUCT
END_TYPE

// DUTs/T_matrix8xdouble
(* Generated from type 'matrix8xdouble' *)
{attribute 'TcIecLibraryType'}
TYPE T_matrix8xdouble : ARRAY [0..7] OF LREAL;
END_TYPE

// DUTs/T_matrix8x4xdouble
(* Generated from type 'matrix8x4xdouble' *)
{attribute 'TcIecLibraryType'}
TYPE T_matrix8x4xdouble : ARRAY [0..3,0..7] OF LREAL;
END_TYPE

// DUTs/PLREAL
{attribute 'TcIecLibraryType'}
TYPE PLREAL : POINTER TO LREAL;
END_TYPE

// DUTs/T_matrix4xdoublepointer
(* Generated from type 'matrix4xdouble *' *)
{attribute 'TcIecLibraryType'}
{attribute 'BaseTypeGUID' := '2CE33DB5-EBD3-49F7-1FA0-F8105FFA7B54'}
TYPE T_matrix4xdoublepointer : ARRAY [0..3] OF PLREAL;
END_TYPE

// DUTs/ST_ODE4_IntgData
(* Generated from type 'ODE4_IntgData' *)
{attribute 'TcIecLibraryType'}
{attribute 'pack_mode' := '1'}
TYPE ST_ODE4_IntgData : 
	STRUCT
		y : POINTER TO LREAL;
		(* Generated from item 'f' *)
		af : T_matrix4xdoublepointer;
	END_STRUCT
END_TYPE

// DUTs/ST_DW_lateral_levitation_control_new_T
(* Generated from type 'DW_lateral_levitation_control_new_T' *)
{attribute 'TcIecLibraryType'}
TYPE ST_DW_lateral_levitation_control_new_T : 
	STRUCT
		(* Generated from item 'UnitDelay_DSTATE' *)
		aUnitDelay_DSTATE : T_matrix2xdouble;
		(* Generated from item 'UnitDelay1_DSTATE' *)
		fUnitDelay1_DSTATE : LREAL;
		(* Generated from item 'UnitDelay1_DSTATE_a' *)
		fUnitDelay1_DSTATE_a : LREAL;
		(* Generated from item 'UnitDelay1_DSTATE_e' *)
		fUnitDelay1_DSTATE_e : LREAL;
		(* Generated from item 'UnitDelay1_DSTATE_c' *)
		fUnitDelay1_DSTATE_c : LREAL;
		(* Generated from item 'UnitDelay1_DSTATE_p' *)
		fUnitDelay1_DSTATE_p : LREAL;
		(* Generated from item 'UnitDelay1_DSTATE_ew' *)
		fUnitDelay1_DSTATE_ew : LREAL;
		(* Generated from item 'UnitDelay1_DSTATE_ce' *)
		fUnitDelay1_DSTATE_ce : LREAL;
		(* Generated from item 'UnitDelay1_DSTATE_f' *)
		fUnitDelay1_DSTATE_f : LREAL;
		(* Generated from item 'UnitDelay1_DSTATE_ez' *)
		fUnitDelay1_DSTATE_ez : LREAL;
		(* Generated from item 'UnitDelay1_DSTATE_b' *)
		fUnitDelay1_DSTATE_b : LREAL;
		(* Generated from item 'UnitDelay1_DSTATE_i' *)
		fUnitDelay1_DSTATE_i : LREAL;
		(* Generated from item 'UnitDelay1_DSTATE_j' *)
		fUnitDelay1_DSTATE_j : LREAL;
		(* Generated from item 'UnitDelay1_DSTATE_o' *)
		fUnitDelay1_DSTATE_o : LREAL;
		(* Generated from item 'UnitDelay1_DSTATE_iw' *)
		fUnitDelay1_DSTATE_iw : LREAL;
		(* Generated from item 'UnitDelay2_DSTATE' *)
		fUnitDelay2_DSTATE : LREAL;
		(* Generated from item 'UnitDelay2_DSTATE_c' *)
		fUnitDelay2_DSTATE_c : LREAL;
		(* Generated from item 'UnitDelay2_DSTATE_m' *)
		fUnitDelay2_DSTATE_m : LREAL;
		(* Generated from item 'UnitDelay2_DSTATE_mk' *)
		fUnitDelay2_DSTATE_mk : LREAL;
		(* Generated from item 'UnitDelay2_DSTATE_l' *)
		fUnitDelay2_DSTATE_l : LREAL;
		(* Generated from item 'UnitDelay2_DSTATE_e' *)
		fUnitDelay2_DSTATE_e : LREAL;
		(* Generated from item 'UnitDelay2_DSTATE_o' *)
		fUnitDelay2_DSTATE_o : LREAL;
		(* Generated from item 'UnitDelay2_DSTATE_i' *)
		fUnitDelay2_DSTATE_i : LREAL;
		(* Generated from item 'UnitDelay2_DSTATE_o5' *)
		fUnitDelay2_DSTATE_o5 : LREAL;
		(* Generated from item 'UnitDelay2_DSTATE_h' *)
		fUnitDelay2_DSTATE_h : LREAL;
		(* Generated from item 'UnitDelay2_DSTATE_b' *)
		fUnitDelay2_DSTATE_b : LREAL;
		(* Generated from item 'UnitDelay2_DSTATE_ej' *)
		fUnitDelay2_DSTATE_ej : LREAL;
		(* Generated from item 'UnitDelay2_DSTATE_eo' *)
		fUnitDelay2_DSTATE_eo : LREAL;
		(* Generated from item 'UnitDelay2_DSTATE_o1' *)
		fUnitDelay2_DSTATE_o1 : LREAL;
	END_STRUCT
END_TYPE

// DUTs/ST_x08a7a7bbd0e5d629f7d70ceec84eacfe
(* Generated from type 'x08a7a7bbd0e5d629f7d70ceec84eacfe' *)
{attribute 'TcIecLibraryType'}
TYPE ST_x08a7a7bbd0e5d629f7d70ceec84eacfe : 
	STRUCT
		(* Generated from item 'numContStates' *)
		nnumContStates : DINT;
		(* Generated from item 'numPeriodicContStates' *)
		nnumPeriodicContStates : DINT;
		(* Generated from item 'numSampTimes' *)
		nnumSampTimes : DINT;
	END_STRUCT
END_TYPE

// DUTs/ST_xf09845edab6c83520d8d57def6d6fe1c
(* Generated from type 'xf09845edab6c83520d8d57def6d6fe1c' *)
{attribute 'TcIecLibraryType'}
TYPE ST_xf09845edab6c83520d8d57def6d6fe1c : 
	STRUCT
		(* Generated from item 'clockTick0' *)
		nclockTick0 : UDINT;
		(* Generated from item 'clockTickH0' *)
		nclockTickH0 : UDINT;
		(* Generated from item 'stepSize0' *)
		fstepSize0 : LREAL;
		(* Generated from item 'clockTick1' *)
		nclockTick1 : UDINT;
		(* Generated from item 'clockTickH1' *)
		nclockTickH1 : UDINT;
		(* Generated from item 'tStart' *)
		ftStart : LREAL;
		(* Generated from item 'simTimeStep' *)
		esimTimeStep : E_SimTimeStep;
		(* Generated from item 'stopRequestedFlag' *)
		bstopRequestedFlag : BOOL;
		 {attribute 'hide'}
		_reserved1 : ARRAY [1..3] OF USINT;
		t : POINTER TO LREAL;
		(* Generated from item 'tArray' *)
		atArray : T_matrix2xdouble;
	END_STRUCT
END_TYPE

// DUTs/ST_RT_MODEL_lateral_levitation_control_new_T
(* Generated from type 'RT_MODEL_lateral_levitation_control_new_T' *)
{attribute 'TcIecLibraryType'}
{attribute 'pack_mode' := '1'}
TYPE ST_RT_MODEL_lateral_levitation_control_new_T : 
	STRUCT
		errorStatus : POINTER TO SINT;
		solverInfo : POINTER TO ST_ssSolverInfo;
		blockIO : POINTER TO ST_B_lateral_levitation_control_new_T;
		prevZCSigState : POINTER TO ST_PrevZCX_lateral_levitation_control_new_T;
		contStates : POINTER TO ST_X_lateral_levitation_control_new_T;
		periodicContStateIndices : POINTER TO DINT;
		periodicContStateRanges : POINTER TO LREAL;
		derivs : POINTER TO LREAL;
		inputs : POINTER TO ST_ExtU_lateral_levitation_control_new_T;
		outputs : POINTER TO ST_ExtY_lateral_levitation_control_new_T;
		contStateDisabled : POINTER TO ST_XDis_lateral_levitation_control_new_T;
		(* Generated from item 'zCCacheNeedsReset' *)
		bzCCacheNeedsReset : BOOL;
		(* Generated from item 'derivCacheNeedsReset' *)
		bderivCacheNeedsReset : BOOL;
		(* Generated from item 'CTOutputIncnstWithState' *)
		bCTOutputIncnstWithState : BOOL;
		 {attribute 'hide'}
		_reserved1 : UINT_8_40;
		(* Generated from item 'odeY' *)
		aodeY : T_matrix8xdouble;
		(* Generated from item 'odeF' *)
		aodeF : T_matrix8x4xdouble;
		(* Generated from item 'intgData' *)
		stintgData : ST_ODE4_IntgData;
		dwork : POINTER TO ST_DW_lateral_levitation_control_new_T;
		(* Generated from item 'Sizes' *)
		stSizes : ST_x08a7a7bbd0e5d629f7d70ceec84eacfe;
		 {attribute 'hide'}
		_reserved2 : UDINT;
		(* Generated from item 'Timing' *)
		stTiming : ST_xf09845edab6c83520d8d57def6d6fe1c;
	END_STRUCT
END_TYPE

// DUTs/T_matrix14xdouble
(* Generated from type 'matrix14xdouble' *)
{attribute 'TcIecLibraryType'}
TYPE T_matrix14xdouble : ARRAY [0..13] OF LREAL;
END_TYPE

// DUTs/T_matrix112xdouble
(* Generated from type 'matrix112xdouble' *)
{attribute 'TcIecLibraryType'}
TYPE T_matrix112xdouble : ARRAY [0..111] OF LREAL;
END_TYPE

// DUTs/ST_P_lateral_levitation_control_new_T
(* Generated from type 'P_lateral_levitation_control_new_T' *)
{attribute 'TcIecLibraryType'}
TYPE ST_P_lateral_levitation_control_new_T : 
	STRUCT
		(* Generated from item 'Is_ems' *)
		aIs_ems : T_matrix14xdouble;
		(* Generated from item 'K_D_lat' *)
		fK_D_lat : LREAL;
		(* Generated from item 'K_D_yaw' *)
		fK_D_yaw : LREAL;
		(* Generated from item 'K_F_init_lat' *)
		fK_F_init_lat : LREAL;
		(* Generated from item 'K_F_init_yaw' *)
		fK_F_init_yaw : LREAL;
		(* Generated from item 'K_F_lat' *)
		fK_F_lat : LREAL;
		(* Generated from item 'K_F_yaw' *)
		fK_F_yaw : LREAL;
		(* Generated from item 'K_I_init_lat' *)
		fK_I_init_lat : LREAL;
		(* Generated from item 'K_I_init_yaw' *)
		fK_I_init_yaw : LREAL;
		(* Generated from item 'K_I_lat' *)
		fK_I_lat : LREAL;
		(* Generated from item 'K_I_yaw' *)
		fK_I_yaw : LREAL;
		(* Generated from item 'K_P_lat' *)
		fK_P_lat : LREAL;
		(* Generated from item 'K_P_yaw' *)
		fK_P_yaw : LREAL;
		(* Generated from item 'airgap_nominal_ems' *)
		fairgap_nominal_ems : LREAL;
		(* Generated from item 'd_EMS_to_EMS' *)
		fd_EMS_to_EMS : LREAL;
		(* Generated from item 'ems_under_gap' *)
		fems_under_gap : LREAL;
		(* Generated from item 'f_extra_y_filter_1' *)
		ff_extra_y_filter_1 : LREAL;
		(* Generated from item 'f_extra_y_filter_2' *)
		ff_extra_y_filter_2 : LREAL;
		(* Generated from item 'f_extra_y_filter_3' *)
		ff_extra_y_filter_3 : LREAL;
		(* Generated from item 'f_extra_yaw_filter_1' *)
		ff_extra_yaw_filter_1 : LREAL;
		(* Generated from item 'f_extra_yaw_filter_2' *)
		ff_extra_yaw_filter_2 : LREAL;
		(* Generated from item 'f_extra_yaw_filter_3' *)
		ff_extra_yaw_filter_3 : LREAL;
		(* Generated from item 'f_lat_notch_main_1' *)
		ff_lat_notch_main_1 : LREAL;
		(* Generated from item 'f_lat_notch_main_2' *)
		ff_lat_notch_main_2 : LREAL;
		(* Generated from item 'f_lat_notch_main_3' *)
		ff_lat_notch_main_3 : LREAL;
		(* Generated from item 'f_lat_notch_main_4' *)
		ff_lat_notch_main_4 : LREAL;
		(* Generated from item 'force_table_ems' *)
		aforce_table_ems : T_matrix112xdouble;
		(* Generated from item 'motor_y_gain' *)
		fmotor_y_gain : LREAL;
		(* Generated from item 'motor_yaw_gain' *)
		fmotor_yaw_gain : LREAL;
		(* Generated from item 'notch_damp' *)
		fnotch_damp : LREAL;
		(* Generated from item 'notch_gmin' *)
		fnotch_gmin : LREAL;
		(* Generated from item 'r_motor_left_com' *)
		ar_motor_left_com : T_matrix3xdouble;
		(* Generated from item 'r_motor_right_com' *)
		ar_motor_right_com : T_matrix3xdouble;
		(* Generated from item 'r_yaw' *)
		fr_yaw : LREAL;
		(* Generated from item 'r_yaw_ems' *)
		ar_yaw_ems : T_matrix4xdouble;
		(* Generated from item 'thermal_gap_gain_ems' *)
		fthermal_gap_gain_ems : LREAL;
		(* Generated from item 'wheel_compression_liftoff' *)
		fwheel_compression_liftoff : LREAL;
		(* Generated from item 'xs_ems' *)
		axs_ems : T_matrix8xdouble;
		(* Generated from item 'y_target' *)
		fy_target : LREAL;
		(* Generated from item 'yaw_target' *)
		fyaw_target : LREAL;
		(* Generated from item 'z_com' *)
		fz_com : LREAL;
		(* Generated from item 'z_initial_lift_off' *)
		fz_initial_lift_off : LREAL;
		(* Generated from item 'enable_extra_y_notch_1' *)
		benable_extra_y_notch_1 : BOOL;
		(* Generated from item 'enable_extra_y_notch_2' *)
		benable_extra_y_notch_2 : BOOL;
		(* Generated from item 'enable_extra_y_notch_3' *)
		benable_extra_y_notch_3 : BOOL;
		(* Generated from item 'enable_extra_yaw_notch_1' *)
		benable_extra_yaw_notch_1 : BOOL;
		(* Generated from item 'enable_extra_yaw_notch_2' *)
		benable_extra_yaw_notch_2 : BOOL;
		(* Generated from item 'enable_extra_yaw_notch_3' *)
		benable_extra_yaw_notch_3 : BOOL;
		(* Generated from item 'enable_lat_main_notch_1' *)
		benable_lat_main_notch_1 : BOOL;
		(* Generated from item 'enable_lat_main_notch_2' *)
		benable_lat_main_notch_2 : BOOL;
		(* Generated from item 'enable_lat_main_notch_3' *)
		benable_lat_main_notch_3 : BOOL;
		(* Generated from item 'enable_lat_main_notch_4' *)
		benable_lat_main_notch_4 : BOOL;
		(* Generated from item 'feed_forward_ems_ON' *)
		bfeed_forward_ems_ON : BOOL;
		(* Generated from item 'feed_fwd_motor_y_ON' *)
		bfeed_fwd_motor_y_ON : BOOL;
		(* Generated from item 'feed_fwd_motor_yaw_ON' *)
		bfeed_fwd_motor_yaw_ON : BOOL;
		(* Generated from item 'levi_operational' *)
		blevi_operational : BOOL;
		(* Generated from item 'y_ON' *)
		by_ON : BOOL;
		(* Generated from item 'yaw_ON' *)
		byaw_ON : BOOL;
		(* Generated from item 'max_peak_current_Value' *)
		fmax_peak_current_Value : LREAL;
		(* Generated from item 'Constant4_Value' *)
		fConstant4_Value : LREAL;
		(* Generated from item 'UnitDelay_InitialCondition' *)
		fUnitDelay_InitialCondition : LREAL;
		(* Generated from item 'Integrator1_IC' *)
		fIntegrator1_IC : LREAL;
		(* Generated from item 'Constant5_Value' *)
		fConstant5_Value : LREAL;
		(* Generated from item 'Switch1_Threshold' *)
		fSwitch1_Threshold : LREAL;
		(* Generated from item 'max_nominal_current_Value' *)
		fmax_nominal_current_Value : LREAL;
		(* Generated from item 'Switch3_Threshold' *)
		fSwitch3_Threshold : LREAL;
		(* Generated from item 'tau_Gain' *)
		ftau_Gain : LREAL;
		(* Generated from item 'Bias_Bias' *)
		fBias_Bias : LREAL;
		(* Generated from item 'two_Gain' *)
		ftwo_Gain : LREAL;
		(* Generated from item 'one_Gain' *)
		fone_Gain : LREAL;
		(* Generated from item 'UnitDelay1_InitialCondition' *)
		fUnitDelay1_InitialCondition : LREAL;
		(* Generated from item 'tau_Gain_j' *)
		ftau_Gain_j : LREAL;
		(* Generated from item 'Bias_Bias_h' *)
		fBias_Bias_h : LREAL;
		(* Generated from item 'two_Gain_o' *)
		ftwo_Gain_o : LREAL;
		(* Generated from item 'one_Gain_h' *)
		fone_Gain_h : LREAL;
		(* Generated from item 'UnitDelay1_InitialCondition_i' *)
		fUnitDelay1_InitialCondition_i : LREAL;
		(* Generated from item 'tau_Gain_a' *)
		ftau_Gain_a : LREAL;
		(* Generated from item 'Bias_Bias_o' *)
		fBias_Bias_o : LREAL;
		(* Generated from item 'two_Gain_l' *)
		ftwo_Gain_l : LREAL;
		(* Generated from item 'one_Gain_i' *)
		fone_Gain_i : LREAL;
		(* Generated from item 'UnitDelay1_InitialCondition_m' *)
		fUnitDelay1_InitialCondition_m : LREAL;
		(* Generated from item 'tau_Gain_m' *)
		ftau_Gain_m : LREAL;
		(* Generated from item 'Bias_Bias_j' *)
		fBias_Bias_j : LREAL;
		(* Generated from item 'two_Gain_e' *)
		ftwo_Gain_e : LREAL;
		(* Generated from item 'one_Gain_n' *)
		fone_Gain_n : LREAL;
		(* Generated from item 'UnitDelay1_InitialCondition_g' *)
		fUnitDelay1_InitialCondition_g : LREAL;
		(* Generated from item 'tau_Gain_d' *)
		ftau_Gain_d : LREAL;
		(* Generated from item 'Bias_Bias_oz' *)
		fBias_Bias_oz : LREAL;
		(* Generated from item 'two_Gain_c' *)
		ftwo_Gain_c : LREAL;
		(* Generated from item 'one_Gain_j' *)
		fone_Gain_j : LREAL;
		(* Generated from item 'UnitDelay1_InitialCondition_g4' *)
		fUnitDelay1_InitialCondition_g4 : LREAL;
		(* Generated from item 'tau_Gain_k' *)
		ftau_Gain_k : LREAL;
		(* Generated from item 'Bias_Bias_k' *)
		fBias_Bias_k : LREAL;
		(* Generated from item 'two_Gain_f' *)
		ftwo_Gain_f : LREAL;
		(* Generated from item 'one_Gain_p' *)
		fone_Gain_p : LREAL;
		(* Generated from item 'UnitDelay1_InitialCondition_l' *)
		fUnitDelay1_InitialCondition_l : LREAL;
		(* Generated from item 'tau_Gain_g' *)
		ftau_Gain_g : LREAL;
		(* Generated from item 'Bias_Bias_m' *)
		fBias_Bias_m : LREAL;
		(* Generated from item 'two_Gain_ek' *)
		ftwo_Gain_ek : LREAL;
		(* Generated from item 'one_Gain_b' *)
		fone_Gain_b : LREAL;
		(* Generated from item 'UnitDelay1_InitialCondition_iv' *)
		fUnitDelay1_InitialCondition_iv : LREAL;
		(* Generated from item 'tau_Gain_e' *)
		ftau_Gain_e : LREAL;
		(* Generated from item 'Bias_Bias_i' *)
		fBias_Bias_i : LREAL;
		(* Generated from item 'two_Gain_h' *)
		ftwo_Gain_h : LREAL;
		(* Generated from item 'one_Gain_g' *)
		fone_Gain_g : LREAL;
		(* Generated from item 'UnitDelay1_InitialCondition_gp' *)
		fUnitDelay1_InitialCondition_gp : LREAL;
		(* Generated from item 'tau_Gain_i' *)
		ftau_Gain_i : LREAL;
		(* Generated from item 'Bias_Bias_kg' *)
		fBias_Bias_kg : LREAL;
		(* Generated from item 'two_Gain_fh' *)
		ftwo_Gain_fh : LREAL;
		(* Generated from item 'one_Gain_bj' *)
		fone_Gain_bj : LREAL;
		(* Generated from item 'UnitDelay1_InitialCondition_iq' *)
		fUnitDelay1_InitialCondition_iq : LREAL;
		(* Generated from item 'tau_Gain_ko' *)
		ftau_Gain_ko : LREAL;
		(* Generated from item 'Bias_Bias_e' *)
		fBias_Bias_e : LREAL;
		(* Generated from item 'two_Gain_j' *)
		ftwo_Gain_j : LREAL;
		(* Generated from item 'one_Gain_o' *)
		fone_Gain_o : LREAL;
		(* Generated from item 'UnitDelay1_InitialCondition_f' *)
		fUnitDelay1_InitialCondition_f : LREAL;
		(* Generated from item 'tau_Gain_jc' *)
		ftau_Gain_jc : LREAL;
		(* Generated from item 'Bias_Bias_b' *)
		fBias_Bias_b : LREAL;
		(* Generated from item 'two_Gain_hf' *)
		ftwo_Gain_hf : LREAL;
		(* Generated from item 'one_Gain_jm' *)
		fone_Gain_jm : LREAL;
		(* Generated from item 'UnitDelay1_InitialCondition_id' *)
		fUnitDelay1_InitialCondition_id : LREAL;
		(* Generated from item 'tau_Gain_c' *)
		ftau_Gain_c : LREAL;
		(* Generated from item 'Bias_Bias_n' *)
		fBias_Bias_n : LREAL;
		(* Generated from item 'two_Gain_b' *)
		ftwo_Gain_b : LREAL;
		(* Generated from item 'one_Gain_nu' *)
		fone_Gain_nu : LREAL;
		(* Generated from item 'UnitDelay1_InitialCondition_e' *)
		fUnitDelay1_InitialCondition_e : LREAL;
		(* Generated from item 'tau_Gain_n' *)
		ftau_Gain_n : LREAL;
		(* Generated from item 'Bias_Bias_a' *)
		fBias_Bias_a : LREAL;
		(* Generated from item 'two_Gain_c3' *)
		ftwo_Gain_c3 : LREAL;
		(* Generated from item 'one_Gain_f' *)
		fone_Gain_f : LREAL;
		(* Generated from item 'UnitDelay1_InitialCondition_b' *)
		fUnitDelay1_InitialCondition_b : LREAL;
		(* Generated from item 'tau_Gain_ks' *)
		ftau_Gain_ks : LREAL;
		(* Generated from item 'Bias_Bias_m2' *)
		fBias_Bias_m2 : LREAL;
		(* Generated from item 'two_Gain_f3' *)
		ftwo_Gain_f3 : LREAL;
		(* Generated from item 'one_Gain_m' *)
		fone_Gain_m : LREAL;
		(* Generated from item 'UnitDelay1_InitialCondition_eg' *)
		fUnitDelay1_InitialCondition_eg : LREAL;
		(* Generated from item 'Constant_Value' *)
		fConstant_Value : LREAL;
		(* Generated from item 'Gain10_Gain' *)
		fGain10_Gain : LREAL;
		(* Generated from item 'min_peak_current_Value' *)
		fmin_peak_current_Value : LREAL;
		(* Generated from item 'min_nominal_current_Value' *)
		fmin_nominal_current_Value : LREAL;
		(* Generated from item 'Switch4_Threshold' *)
		fSwitch4_Threshold : LREAL;
		(* Generated from item 'Gain20_Gain' *)
		fGain20_Gain : LREAL;
		(* Generated from item 'Bias1_Bias' *)
		fBias1_Bias : LREAL;
		(* Generated from item 'Gain_Gain' *)
		fGain_Gain : LREAL;
		(* Generated from item 'UnitDelay2_InitialCondition' *)
		fUnitDelay2_InitialCondition : LREAL;
		(* Generated from item 'Bias1_Bias_j' *)
		fBias1_Bias_j : LREAL;
		(* Generated from item 'Gain_Gain_a' *)
		fGain_Gain_a : LREAL;
		(* Generated from item 'UnitDelay2_InitialCondition_j' *)
		fUnitDelay2_InitialCondition_j : LREAL;
		(* Generated from item 'Bias1_Bias_i' *)
		fBias1_Bias_i : LREAL;
		(* Generated from item 'Gain_Gain_l' *)
		fGain_Gain_l : LREAL;
		(* Generated from item 'UnitDelay2_InitialCondition_k' *)
		fUnitDelay2_InitialCondition_k : LREAL;
		(* Generated from item 'Bias1_Bias_b' *)
		fBias1_Bias_b : LREAL;
		(* Generated from item 'Gain_Gain_n' *)
		fGain_Gain_n : LREAL;
		(* Generated from item 'UnitDelay2_InitialCondition_a' *)
		fUnitDelay2_InitialCondition_a : LREAL;
		(* Generated from item 'Bias1_Bias_f' *)
		fBias1_Bias_f : LREAL;
		(* Generated from item 'Gain_Gain_ar' *)
		fGain_Gain_ar : LREAL;
		(* Generated from item 'UnitDelay2_InitialCondition_i' *)
		fUnitDelay2_InitialCondition_i : LREAL;
		(* Generated from item 'Bias1_Bias_a' *)
		fBias1_Bias_a : LREAL;
		(* Generated from item 'Gain_Gain_f' *)
		fGain_Gain_f : LREAL;
		(* Generated from item 'UnitDelay2_InitialCondition_p' *)
		fUnitDelay2_InitialCondition_p : LREAL;
		(* Generated from item 'Bias1_Bias_p' *)
		fBias1_Bias_p : LREAL;
		(* Generated from item 'Gain_Gain_g' *)
		fGain_Gain_g : LREAL;
		(* Generated from item 'UnitDelay2_InitialCondition_f' *)
		fUnitDelay2_InitialCondition_f : LREAL;
		(* Generated from item 'Bias1_Bias_pq' *)
		fBias1_Bias_pq : LREAL;
		(* Generated from item 'Gain_Gain_e' *)
		fGain_Gain_e : LREAL;
		(* Generated from item 'UnitDelay2_InitialCondition_c' *)
		fUnitDelay2_InitialCondition_c : LREAL;
		(* Generated from item 'Bias1_Bias_h' *)
		fBias1_Bias_h : LREAL;
		(* Generated from item 'Gain_Gain_ep' *)
		fGain_Gain_ep : LREAL;
		(* Generated from item 'UnitDelay2_InitialCondition_o' *)
		fUnitDelay2_InitialCondition_o : LREAL;
		(* Generated from item 'Bias1_Bias_p4' *)
		fBias1_Bias_p4 : LREAL;
		(* Generated from item 'Gain_Gain_ld' *)
		fGain_Gain_ld : LREAL;
		(* Generated from item 'UnitDelay2_InitialCondition_cr' *)
		fUnitDelay2_InitialCondition_cr : LREAL;
		(* Generated from item 'Bias1_Bias_e' *)
		fBias1_Bias_e : LREAL;
		(* Generated from item 'Gain_Gain_lj' *)
		fGain_Gain_lj : LREAL;
		(* Generated from item 'UnitDelay2_InitialCondition_h' *)
		fUnitDelay2_InitialCondition_h : LREAL;
		(* Generated from item 'Bias1_Bias_bf' *)
		fBias1_Bias_bf : LREAL;
		(* Generated from item 'Gain_Gain_ly' *)
		fGain_Gain_ly : LREAL;
		(* Generated from item 'UnitDelay2_InitialCondition_hx' *)
		fUnitDelay2_InitialCondition_hx : LREAL;
		(* Generated from item 'Bias1_Bias_il' *)
		fBias1_Bias_il : LREAL;
		(* Generated from item 'Gain_Gain_g0' *)
		fGain_Gain_g0 : LREAL;
		(* Generated from item 'UnitDelay2_InitialCondition_ab' *)
		fUnitDelay2_InitialCondition_ab : LREAL;
		(* Generated from item 'Bias1_Bias_bd' *)
		fBias1_Bias_bd : LREAL;
		(* Generated from item 'Gain_Gain_h' *)
		fGain_Gain_h : LREAL;
		(* Generated from item 'UnitDelay2_InitialCondition_hl' *)
		fUnitDelay2_InitialCondition_hl : LREAL;
		(* Generated from item 'Constant1_Value' *)
		fConstant1_Value : LREAL;
		(* Generated from item 'Constant10_Value' *)
		fConstant10_Value : LREAL;
		(* Generated from item 'Constant11_Value' *)
		fConstant11_Value : LREAL;
		(* Generated from item 'Constant2_Value' *)
		fConstant2_Value : LREAL;
		(* Generated from item 'Constant6_Value' *)
		fConstant6_Value : LREAL;
		(* Generated from item 'Integrator2_IC' *)
		fIntegrator2_IC : LREAL;
		(* Generated from item 'IsPeak1_Threshold' *)
		fIsPeak1_Threshold : LREAL;
		(* Generated from item 'Switch2_Threshold' *)
		fSwitch2_Threshold : LREAL;
		(* Generated from item 'Constant2_Value_c' *)
		fConstant2_Value_c : LREAL;
		(* Generated from item 'Constant2_Value_b' *)
		fConstant2_Value_b : LREAL;
	END_STRUCT
END_TYPE

// DUTs/E_ModuleCaller
(* Generated from type 'TcMgSdk.ModuleCaller' *)
{attribute 'TcIecLibraryType'}
TYPE E_ModuleCaller : (
	CyclicTask:=0, 	(* Add to the specified cyclic caller tasks. *)
	Module:=1	(* Don't add to cyclic callers. The module can be called from other TwinCAT modules (e. g. a PLC). *)
) DINT;
END_TYPE

// DUTs/E_CallerVerification
(* Generated from type 'TcMgSdk.CallerVerification' *)
{attribute 'TcIecLibraryType'}
TYPE E_CallerVerification : (
	Default:=0, 	(* Verify the caller task only if the "ModuleCaller" parameter is set to "Module" but not when added to cyclic caller tasks. *)
	Always:=1, 	(* Always verify the caller context to prevent concurrent execution of model code and corresponding DataArea mappings. *)
	Never:=2	(* Skip caller verification to reduce execution times. *)
) DINT;
END_TYPE

// DUTs/E_StepSizeAdaptation
(* Generated from type 'TcMgSdk.StepSizeAdaptation' *)
{attribute 'TcIecLibraryType'}
TYPE E_StepSizeAdaptation : (
	RequireMatchingTaskCycleTime:=0, 	(* Don't accept task cycle times other than the Simulink step sizes. *)
	UseTaskCycleTime:=1, 	(* Adapt the Smulink step sizes to the task cycle times. *)
	UseModelStepSize:=2	(* Keep the Smulink step sizes, independent of the callers cycle time. *)
) DINT;
END_TYPE

// DUTs/E_ExecutionSequence1
(* Generated from type 'TcMgSdk.ExecutionSequence1' *)
{attribute 'TcIecLibraryType'}
TYPE E_ExecutionSequence1 : (
	UpdateBeforeOutputMapping:=0, 	(* Input mapping -> State and output update -> Output mapping -> ADS processing *)
	IoAtTaskBegin:=1	(* Input mapping -> Code execution -> Output update -> ADS processing *)
) DINT;
END_TYPE

// DUTs/E_FpExcptCtrlSet
(* Generated from type 'TcMgSdk.FpExcptCtrlSet' *)
{attribute 'TcIecLibraryType'}
TYPE E_FpExcptCtrlSet : (
	CallerExceptions:=1, 	(* Use the floating point exception settings provided by the caller *)
	ThrowExceptions:=3, 	(* Enable floating point exceptions on invalid operations and divisions by zero *)
	SuppressExceptions:=5	(* Disable floating point exceptions. *)
) USINT;
END_TYPE

// DUTs/ST_TcMatSim_ModuleGeneratorInfo
(* Generated from type 'TcMatSim.ModuleGeneratorInfo' *)
{attribute 'TcIecLibraryType'}
TYPE ST_TcMatSim_ModuleGeneratorInfo : 
	STRUCT
		(* Generated from item 'MatlabVersion' *)
		nMatlabVersion : ARRAY [0..3] OF UDINT;
		(* Generated from item 'TE140xVersion' *)
		nTE140xVersion : ARRAY [0..3] OF UDINT;
	END_STRUCT
END_TYPE

// DUTs/ST_TcMatSim_SimulinkModelInfo
(* Generated from type 'TcMatSim.SimulinkModelInfo' *)
{attribute 'TcIecLibraryType'}
TYPE ST_TcMatSim_SimulinkModelInfo : 
	STRUCT
		(* Generated from item 'ModelName' *)
		{attribute 'GUID' := '18071995-0000-0000-0000-00010000007F'}
		sModelName : STRING(127);
		(* Generated from item 'SimulinkVersion' *)
		nSimulinkVersion : ARRAY [0..3] OF UDINT;
		(* Generated from item 'ModelVersion' *)
		nModelVersion : ARRAY [0..3] OF UDINT;
		(* Generated from item 'ModelChecksum' *)
		nModelChecksum : ARRAY [0..3] OF UDINT;
	END_STRUCT
END_TYPE

// DUTs/E_ParameterSharingType
(* Generated from type 'ParameterSharingType' *)
{attribute 'TcIecLibraryType'}
TYPE E_ParameterSharingType : (
	Define:=0, 	(* This module instance defines the parameter values for all further instances of this module class. Exactly one instance of this module class must use this option. *)
	Inherit:=1	(* This module instance inherits the parameter values from the instance of this module class configured to "Define" the parameter values. Model parameters configured at this instsance are ignored. *)
) DINT;
END_TYPE

// DUTs/ST_FB_lateral_levitation_control_new_TcCOM_InitStruct
{attribute 'TcIecLibraryType'}
TYPE ST_FB_lateral_levitation_control_new_TcCOM_InitStruct : 
	STRUCT
		{attribute 'GUID' := '18071995-0000-0000-0000-000000000061'}
		eObjState : TCOM_STATE := TCOM_STATE.TCOM_STATE_OP;
		{attribute 'GUID' := '18071995-0000-0000-0000-00010000007F'}
		sObjName : STRING(127);
		{attribute 'GUID' := '18071995-0000-0000-0000-00000000000F'}
		nOid : OTCID := 4294967295;
		{attribute 'GUID' := '18071995-0000-0000-0000-00000000000F'}
		nTaskOid : OTCID;
		nTaskSortOrder : UDINT;
		{attribute 'GUID' := '8007AE3B-86BB-40F2-B385-EF87FCC239A4'}
		eTraceLevelMax : TcTraceLevel := TcTraceLevel.tlInfo;
		eModuleCaller : E_ModuleCaller := E_ModuleCaller.CyclicTask;
		eCallerVerification : E_CallerVerification := E_CallerVerification.Default;
		eStepSizeAdaptation : E_StepSizeAdaptation := E_StepSizeAdaptation.RequireMatchingTaskCycleTime;
		eExecutionSequence : E_ExecutionSequence1 := E_ExecutionSequence1.UpdateBeforeOutputMapping;
		bExecute : BOOL := TRUE;
		 {attribute 'hide'}
		_reserved1 : ARRAY [1..3] OF USINT;
		{attribute 'GUID' := '18071995-0000-0000-0000-000000000061'}
		eAccessLockState : TCOM_STATE := TCOM_STATE.TCOM_STATE_OP;
		eInitExceptionHandling : E_FpExcptCtrlSet := E_FpExcptCtrlSet.CallerExceptions;
		eUpdateExceptionHandling : E_FpExcptCtrlSetEx := E_FpExcptCtrlSetEx.CallerExceptions;
		 {attribute 'hide'}
		_reserved2 : UINT;
		stModuleGeneratorInfo : ST_TcMatSim_ModuleGeneratorInfo;
		stSimulinkModelInfo : ST_TcMatSim_SimulinkModelInfo;
		elateral_levitation_control_new_P_Sharing : E_ParameterSharingType := E_ParameterSharingType.Define;
		 {attribute 'hide'}
		_reserved3 : UDINT;
		stlateral_levitation_control_new_P : ST_P_lateral_levitation_control_new_T := (aIs_ems := [0.0,1.0,2.0,3.0,4.0,5.0,6.0,7.0,8.0,9.0,10.0,11.0,12.0,13.0], fK_D_lat := 0, fK_D_yaw := 10000, fK_F_init_lat := 0, fK_F_init_yaw := 0, fK_F_lat := 0, fK_F_yaw := 100, fK_I_init_lat := 0, fK_I_init_yaw := 0, fK_I_lat := 0, fK_I_yaw := 4000, fK_P_lat := 0, fK_P_yaw := 300000, fairgap_nominal_ems := 0.008, fd_EMS_to_EMS := 0.32, fems_under_gap := 0, ff_extra_y_filter_1 := 50.66, ff_extra_y_filter_2 := 50.66, ff_extra_y_filter_3 := 50.66, ff_extra_yaw_filter_1 := 50.66, ff_extra_yaw_filter_2 := 50.66, ff_extra_yaw_filter_3 := 50.66, ff_lat_notch_main_1 := 54.0540540541, ff_lat_notch_main_2 := 41.58, ff_lat_notch_main_3 := 42.86, ff_lat_notch_main_4 := 210.94, aforce_table_ems := [-0,-0,-0,-0,-0,-0,-0,-0,655.13,174.16,81.659,47.261,30.593,21.524,15.713,11.96,2611.6,696.59,326.58,189.04,122.37,86.096,62.854,47.842,5533.7,1564.3,734.24,425.32,275.32,193.71,141.42,107.62,7454.5,2760.2,1303.6,754.96,488.92,344.0,251.18,191.23,8748.8,4055.3,2029.2,1177.9,763.29,537.14,392.24,298.63,9740.3,5057.0,2856.8,1689.8,1097.4,772.66,564.41,429.74,10473.0,5869.3,3587.3,2256.1,1487.3,1049.3,767.15,584.27,11080.0,6542.1,4206.5,2772.3,1900.4,1360.7,998.69,761.45,11592.0,7076.8,4756.5,3227.3,2279.5,1670.0,1246.3,957.29,12028.0,7546.1,5205.9,3645.9,2622.5,1955.5,1481.6,1152.2,12442.0,7965.7,5589.9,4001.4,2944.8,2217.7,1700.9,1335.7,12817.0,8338.4,5942.3,4304.2,3222.4,2466.8,1907.6,1506.7,13127.0,8698.2,6260.2,4584.5,3461.7,2679.6,2098.8,1672.7], fmotor_y_gain := 1, fmotor_yaw_gain := 1, fnotch_damp := 0.3, fnotch_gmin := 0.1, ar_motor_left_com := [0.0147302,0.8070598,0.34816], ar_motor_right_com := [0.0147302,-0.7979402,0.34816], fr_yaw := 0.87325, ar_yaw_ems := [0.8879802,0.8879802,0.8585198,0.8585198], fthermal_gap_gain_ems := 1.16, fwheel_compression_liftoff := 0.0015, axs_ems := [0.002,0.004,0.006,0.008,0.01,0.012,0.014,0.016], fy_target := 0, fyaw_target := 0, fz_com := 0.5706599999999999, fz_initial_lift_off := -0.023, benable_extra_y_notch_1 := FALSE, benable_extra_y_notch_2 := FALSE, benable_extra_y_notch_3 := FALSE, benable_extra_yaw_notch_1 := FALSE, benable_extra_yaw_notch_2 := FALSE, benable_extra_yaw_notch_3 := FALSE, benable_lat_main_notch_1 := TRUE, benable_lat_main_notch_2 := FALSE, benable_lat_main_notch_3 := FALSE, benable_lat_main_notch_4 := FALSE, bfeed_forward_ems_ON := FALSE, bfeed_fwd_motor_y_ON := FALSE, bfeed_fwd_motor_yaw_ON := FALSE, blevi_operational := FALSE, by_ON := TRUE, byaw_ON := TRUE, fmax_peak_current_Value := 10, fConstant4_Value := 0, fUnitDelay_InitialCondition := 0, fIntegrator1_IC := 0, fConstant5_Value := 1, fSwitch1_Threshold := 7, fmax_nominal_current_Value := 4.5, fSwitch3_Threshold := 0, ftau_Gain := 0.00075, fBias_Bias := 1, ftwo_Gain := 2, fone_Gain := 1, fUnitDelay1_InitialCondition := 0, ftau_Gain_j := 0.00075, fBias_Bias_h := 1, ftwo_Gain_o := 2, fone_Gain_h := 1, fUnitDelay1_InitialCondition_i := 0, ftau_Gain_a := 0.00075, fBias_Bias_o := 1, ftwo_Gain_l := 2, fone_Gain_i := 1, fUnitDelay1_InitialCondition_m := 0, ftau_Gain_m := 0.00075, fBias_Bias_j := 1, ftwo_Gain_e := 2, fone_Gain_n := 1, fUnitDelay1_InitialCondition_g := 0, ftau_Gain_d := 0.00075, fBias_Bias_oz := 1, ftwo_Gain_c := 2, fone_Gain_j := 1, fUnitDelay1_InitialCondition_g4 := 0, ftau_Gain_k := 0.00075, fBias_Bias_k := 1, ftwo_Gain_f := 2, fone_Gain_p := 1, fUnitDelay1_InitialCondition_l := 0, ftau_Gain_g := 0.00075, fBias_Bias_m := 1, ftwo_Gain_ek := 2, fone_Gain_b := 1, fUnitDelay1_InitialCondition_iv := 0, ftau_Gain_e := 0.00075, fBias_Bias_i := 1, ftwo_Gain_h := 2, fone_Gain_g := 1, fUnitDelay1_InitialCondition_gp := 0, ftau_Gain_i := 0.00075, fBias_Bias_kg := 1, ftwo_Gain_fh := 2, fone_Gain_bj := 1, fUnitDelay1_InitialCondition_iq := 0, ftau_Gain_ko := 0.00075, fBias_Bias_e := 1, ftwo_Gain_j := 2, fone_Gain_o := 1, fUnitDelay1_InitialCondition_f := 0, ftau_Gain_jc := 0.00075, fBias_Bias_b := 1, ftwo_Gain_hf := 2, fone_Gain_jm := 1, fUnitDelay1_InitialCondition_id := 0, ftau_Gain_c := 0.00075, fBias_Bias_n := 1, ftwo_Gain_b := 2, fone_Gain_nu := 1, fUnitDelay1_InitialCondition_e := 0, ftau_Gain_n := 0.00075, fBias_Bias_a := 1, ftwo_Gain_c3 := 2, fone_Gain_f := 1, fUnitDelay1_InitialCondition_b := 0, ftau_Gain_ks := 0.00075, fBias_Bias_m2 := 1, ftwo_Gain_f3 := 2, fone_Gain_m := 1, fUnitDelay1_InitialCondition_eg := 0, fConstant_Value := 1, fGain10_Gain := -1, fmin_peak_current_Value := -10, fmin_nominal_current_Value := -4.5, fSwitch4_Threshold := 0, fGain20_Gain := -1, fBias1_Bias := 1, fGain_Gain := 2, fUnitDelay2_InitialCondition := 0, fBias1_Bias_j := 1, fGain_Gain_a := 2, fUnitDelay2_InitialCondition_j := 0, fBias1_Bias_i := 1, fGain_Gain_l := 2, fUnitDelay2_InitialCondition_k := 0, fBias1_Bias_b := 1, fGain_Gain_n := 2, fUnitDelay2_InitialCondition_a := 0, fBias1_Bias_f := 1, fGain_Gain_ar := 2, fUnitDelay2_InitialCondition_i := 0, fBias1_Bias_a := 1, fGain_Gain_f := 2, fUnitDelay2_InitialCondition_p := 0, fBias1_Bias_p := 1, fGain_Gain_g := 2, fUnitDelay2_InitialCondition_f := 0, fBias1_Bias_pq := 1, fGain_Gain_e := 2, fUnitDelay2_InitialCondition_c := 0, fBias1_Bias_h := 1, fGain_Gain_ep := 2, fUnitDelay2_InitialCondition_o := 0, fBias1_Bias_p4 := 1, fGain_Gain_ld := 2, fUnitDelay2_InitialCondition_cr := 0, fBias1_Bias_e := 1, fGain_Gain_lj := 2, fUnitDelay2_InitialCondition_h := 0, fBias1_Bias_bf := 1, fGain_Gain_ly := 2, fUnitDelay2_InitialCondition_hx := 0, fBias1_Bias_il := 1, fGain_Gain_g0 := 2, fUnitDelay2_InitialCondition_ab := 0, fBias1_Bias_bd := 1, fGain_Gain_h := 2, fUnitDelay2_InitialCondition_hl := 0, fConstant1_Value := 0, fConstant10_Value := 1, fConstant11_Value := 0, fConstant2_Value := 1, fConstant6_Value := 1, fIntegrator2_IC := 0, fIsPeak1_Threshold := 4.5, fSwitch2_Threshold := 7, fConstant2_Value_c := 0, fConstant2_Value_b := 0);
	END_STRUCT
END_TYPE

// DUTs/ST_FB_lateral_levitation_control_new_TcCOM_InitStruct_FB_init
{attribute 'TcIecLibraryType'}
{attribute 'hide'}
TYPE ST_FB_lateral_levitation_control_new_TcCOM_InitStruct_FB_init : 
	STRUCT
		{attribute 'GUID' := '18071995-0000-0000-0000-000000000018'}
		pInst : PVOID;
		bInitRetains : BOOL;
		bInCopyCode : BOOL;
		 {attribute 'hide'}
		_reserved1 : UINT_16_48;
		stInit : REFERENCE TO ST_FB_lateral_levitation_control_new_TcCOM_InitStruct;
		result : BOOL;
		 {attribute 'hide'}
		_reserved2 : UINT_24_56;
	END_STRUCT
END_TYPE

// DUTs/ST_FB_lateral_levitation_control_new_TcCOM_InitStruct_FB_afterinit
{attribute 'TcIecLibraryType'}
{attribute 'hide'}
TYPE ST_FB_lateral_levitation_control_new_TcCOM_InitStruct_FB_afterinit : 
	STRUCT
		{attribute 'GUID' := '18071995-0000-0000-0000-000000000018'}
		pInst : PVOID;
		result : BOOL;
		 {attribute 'hide'}
		_reserved1 : UINT_24_56;
	END_STRUCT
END_TYPE

// DUTs/ST_FB_lateral_levitation_control_new_TcCOM_InitStruct_Reinit
{attribute 'TcIecLibraryType'}
{attribute 'hide'}
TYPE ST_FB_lateral_levitation_control_new_TcCOM_InitStruct_Reinit : 
	STRUCT
		{attribute 'GUID' := '18071995-0000-0000-0000-000000000018'}
		pInst : PVOID;
		stReInit : ST_FB_lateral_levitation_control_new_TcCOM_InitStruct;
		result : BOOL;
		 {attribute 'hide'}
		_reserved1 : ARRAY [1..7] OF USINT;
	END_STRUCT
END_TYPE

// DUTs/ST_FB_lateral_levitation_control_new_TcCOM_InitStruct_FB_Main
{attribute 'TcIecLibraryType'}
{attribute 'hide'}
TYPE ST_FB_lateral_levitation_control_new_TcCOM_InitStruct_FB_Main : 
	STRUCT
		{attribute 'GUID' := '18071995-0000-0000-0000-000000000018'}
		pInst : PVOID;
		result : BOOL;
		 {attribute 'hide'}
		_reserved1 : UINT_24_56;
	END_STRUCT
END_TYPE

// DUTs/ST_FB_lateral_levitation_control_new_TcCOM_InitStruct_FB_exit
{attribute 'TcIecLibraryType'}
{attribute 'hide'}
TYPE ST_FB_lateral_levitation_control_new_TcCOM_InitStruct_FB_exit : 
	STRUCT
		{attribute 'GUID' := '18071995-0000-0000-0000-000000000018'}
		pInst : PVOID;
		bInCopyCode : BOOL;
		result : BOOL;
		 {attribute 'hide'}
		_reserved1 : UINT_16_48;
	END_STRUCT
END_TYPE

// DUTs/ST_GetSet_TCOM_STATE
{attribute 'TcIecLibraryType'}
{attribute 'hide'}
TYPE ST_GetSet_TCOM_STATE : 
	STRUCT
		{attribute 'GUID' := '18071995-0000-0000-0000-000000000018'}
		pInst : PVOID;
		{attribute 'GUID' := '18071995-0000-0000-0000-000000000061'}
		eParam : TCOM_STATE;
		 {attribute 'hide'}
		_reserved1 : UINT_0_32;
	END_STRUCT
END_TYPE

// DUTs/ST_GetSet_ITComObject
{attribute 'TcIecLibraryType'}
{attribute 'hide'}
TYPE ST_GetSet_ITComObject : 
	STRUCT
		{attribute 'GUID' := '18071995-0000-0000-0000-000000000018'}
		pInst : PVOID;
		{attribute 'GUID' := '00000012-0000-0000-E000-000000000064'}
		ipParam : ITComObject;
	END_STRUCT
END_TYPE

// DUTs/ST_GetSet_ITcADI
{attribute 'TcIecLibraryType'}
{attribute 'hide'}
TYPE ST_GetSet_ITcADI : 
	STRUCT
		{attribute 'GUID' := '18071995-0000-0000-0000-000000000018'}
		pInst : PVOID;
		{attribute 'GUID' := '03000012-0000-0000-E000-000000000064'}
		ipParam : ITcADI;
	END_STRUCT
END_TYPE

// DUTs/ST_lateral_levitation_control_new_U_T
(* Generated from type 'lateral_levitation_control_new_U_T' *)
{attribute 'TcIecLibraryType'}
TYPE ST_lateral_levitation_control_new_U_T : 
	STRUCT
		(* Generated from item 'y' *)
		fy : LREAL;
		(* Generated from item 'yaw' *)
		fyaw : LREAL;
		(* Generated from item 'motor_Fx_l' *)
		fmotor_Fx_l : LREAL;
		(* Generated from item 'motor_Fx_r' *)
		fmotor_Fx_r : LREAL;
		(* Generated from item 'motor_Fy_l' *)
		fmotor_Fy_l : LREAL;
		(* Generated from item 'motor_Fy_r' *)
		fmotor_Fy_r : LREAL;
		(* Generated from item 'z' *)
		fz : LREAL;
	END_STRUCT
END_TYPE

// DUTs/ST_lateral_levitation_control_new_Y_T
(* Generated from type 'lateral_levitation_control_new_Y_T' *)
{attribute 'TcIecLibraryType'}
TYPE ST_lateral_levitation_control_new_Y_T : 
	STRUCT
		(* Generated from item 'F_latreq' *)
		aF_latreq : T_matrix2xdouble;
		(* Generated from item 'I_ems' *)
		aI_ems : T_matrix4xdouble;
		(* Generated from item 'F_emsfb' *)
		aF_emsfb : T_matrix2xdouble;
		(* Generated from item 'airgaps' *)
		aairgaps : T_matrix4xdouble;
		(* Generated from item 'integrals' *)
		aintegrals : T_matrix2xdouble;
		(* Generated from item 't_peak' *)
		at_peak : T_matrix2xdouble;
		(* Generated from item 'tau_x_ems' *)
		ftau_x_ems : LREAL;
	END_STRUCT
END_TYPE

// DUTs/ST_lateral_levitation_control_new_X_T
(* Generated from type 'lateral_levitation_control_new_X_T' *)
{attribute 'TcIecLibraryType'}
TYPE ST_lateral_levitation_control_new_X_T : 
	STRUCT
		(* Generated from item 'Integrator_CSTATE' *)
		fIntegrator_CSTATE : LREAL;
		(* Generated from item 'Filtertot_CSTATE' *)
		fFiltertot_CSTATE : LREAL;
		(* Generated from item 'Integrator_CSTATE_d' *)
		fIntegrator_CSTATE_d : LREAL;
		(* Generated from item 'Filtertot_CSTATE_p' *)
		fFiltertot_CSTATE_p : LREAL;
		(* Generated from item 'Integrator1_CSTATE' *)
		aIntegrator1_CSTATE : T_matrix2xdouble;
		(* Generated from item 'Integrator2_CSTATE' *)
		aIntegrator2_CSTATE : T_matrix2xdouble;
	END_STRUCT
END_TYPE

// DUTs/ST_lateral_levitation_control_new_DW_T
(* Generated from type 'lateral_levitation_control_new_DW_T' *)
{attribute 'TcIecLibraryType'}
TYPE ST_lateral_levitation_control_new_DW_T : 
	STRUCT
		(* Generated from item 'UnitDelay_DSTATE' *)
		aUnitDelay_DSTATE : T_matrix2xdouble;
		(* Generated from item 'UnitDelay1_DSTATE' *)
		fUnitDelay1_DSTATE : LREAL;
		(* Generated from item 'UnitDelay1_DSTATE_a' *)
		fUnitDelay1_DSTATE_a : LREAL;
		(* Generated from item 'UnitDelay1_DSTATE_e' *)
		fUnitDelay1_DSTATE_e : LREAL;
		(* Generated from item 'UnitDelay1_DSTATE_c' *)
		fUnitDelay1_DSTATE_c : LREAL;
		(* Generated from item 'UnitDelay1_DSTATE_p' *)
		fUnitDelay1_DSTATE_p : LREAL;
		(* Generated from item 'UnitDelay1_DSTATE_ew' *)
		fUnitDelay1_DSTATE_ew : LREAL;
		(* Generated from item 'UnitDelay1_DSTATE_ce' *)
		fUnitDelay1_DSTATE_ce : LREAL;
		(* Generated from item 'UnitDelay1_DSTATE_f' *)
		fUnitDelay1_DSTATE_f : LREAL;
		(* Generated from item 'UnitDelay1_DSTATE_ez' *)
		fUnitDelay1_DSTATE_ez : LREAL;
		(* Generated from item 'UnitDelay1_DSTATE_b' *)
		fUnitDelay1_DSTATE_b : LREAL;
		(* Generated from item 'UnitDelay1_DSTATE_i' *)
		fUnitDelay1_DSTATE_i : LREAL;
		(* Generated from item 'UnitDelay1_DSTATE_j' *)
		fUnitDelay1_DSTATE_j : LREAL;
		(* Generated from item 'UnitDelay1_DSTATE_o' *)
		fUnitDelay1_DSTATE_o : LREAL;
		(* Generated from item 'UnitDelay1_DSTATE_iw' *)
		fUnitDelay1_DSTATE_iw : LREAL;
		(* Generated from item 'UnitDelay2_DSTATE' *)
		fUnitDelay2_DSTATE : LREAL;
		(* Generated from item 'UnitDelay2_DSTATE_c' *)
		fUnitDelay2_DSTATE_c : LREAL;
		(* Generated from item 'UnitDelay2_DSTATE_m' *)
		fUnitDelay2_DSTATE_m : LREAL;
		(* Generated from item 'UnitDelay2_DSTATE_mk' *)
		fUnitDelay2_DSTATE_mk : LREAL;
		(* Generated from item 'UnitDelay2_DSTATE_l' *)
		fUnitDelay2_DSTATE_l : LREAL;
		(* Generated from item 'UnitDelay2_DSTATE_e' *)
		fUnitDelay2_DSTATE_e : LREAL;
		(* Generated from item 'UnitDelay2_DSTATE_o' *)
		fUnitDelay2_DSTATE_o : LREAL;
		(* Generated from item 'UnitDelay2_DSTATE_i' *)
		fUnitDelay2_DSTATE_i : LREAL;
		(* Generated from item 'UnitDelay2_DSTATE_o5' *)
		fUnitDelay2_DSTATE_o5 : LREAL;
		(* Generated from item 'UnitDelay2_DSTATE_h' *)
		fUnitDelay2_DSTATE_h : LREAL;
		(* Generated from item 'UnitDelay2_DSTATE_b' *)
		fUnitDelay2_DSTATE_b : LREAL;
		(* Generated from item 'UnitDelay2_DSTATE_ej' *)
		fUnitDelay2_DSTATE_ej : LREAL;
		(* Generated from item 'UnitDelay2_DSTATE_eo' *)
		fUnitDelay2_DSTATE_eo : LREAL;
		(* Generated from item 'UnitDelay2_DSTATE_o1' *)
		fUnitDelay2_DSTATE_o1 : LREAL;
	END_STRUCT
END_TYPE

// DUTs/ST_GetSet_OTCID
{attribute 'TcIecLibraryType'}
{attribute 'hide'}
TYPE ST_GetSet_OTCID : 
	STRUCT
		{attribute 'GUID' := '18071995-0000-0000-0000-000000000018'}
		pInst : PVOID;
		{attribute 'GUID' := '18071995-0000-0000-0000-00000000000F'}
		nParam : OTCID;
		 {attribute 'hide'}
		_reserved1 : UINT_0_32;
	END_STRUCT
END_TYPE

// DUTs/ST_GetSet_UDINT
{attribute 'TcIecLibraryType'}
{attribute 'hide'}
TYPE ST_GetSet_UDINT : 
	STRUCT
		{attribute 'GUID' := '18071995-0000-0000-0000-000000000018'}
		pInst : PVOID;
		nParam : UDINT;
		 {attribute 'hide'}
		_reserved1 : UINT_0_32;
	END_STRUCT
END_TYPE

// DUTs/ST_GetSet_UINT
{attribute 'TcIecLibraryType'}
{attribute 'hide'}
TYPE ST_GetSet_UINT : 
	STRUCT
		{attribute 'GUID' := '18071995-0000-0000-0000-000000000018'}
		pInst : PVOID;
		nParam : UINT;
		 {attribute 'hide'}
		_reserved1 : UINT_16_48;
	END_STRUCT
END_TYPE

// DUTs/ST_GetSet_TcTraceLevel
{attribute 'TcIecLibraryType'}
{attribute 'hide'}
TYPE ST_GetSet_TcTraceLevel : 
	STRUCT
		{attribute 'GUID' := '18071995-0000-0000-0000-000000000018'}
		pInst : PVOID;
		{attribute 'GUID' := '8007AE3B-86BB-40F2-B385-EF87FCC239A4'}
		eParam : TcTraceLevel;
		 {attribute 'hide'}
		_reserved1 : UINT_0_32;
	END_STRUCT
END_TYPE

// DUTs/ST_GetSet_E_ModuleCaller
{attribute 'TcIecLibraryType'}
{attribute 'hide'}
TYPE ST_GetSet_E_ModuleCaller : 
	STRUCT
		{attribute 'GUID' := '18071995-0000-0000-0000-000000000018'}
		pInst : PVOID;
		eParam : E_ModuleCaller;
		 {attribute 'hide'}
		_reserved1 : UINT_0_32;
	END_STRUCT
END_TYPE

// DUTs/ST_GetSet_E_CallerVerification
{attribute 'TcIecLibraryType'}
{attribute 'hide'}
TYPE ST_GetSet_E_CallerVerification : 
	STRUCT
		{attribute 'GUID' := '18071995-0000-0000-0000-000000000018'}
		pInst : PVOID;
		eParam : E_CallerVerification;
		 {attribute 'hide'}
		_reserved1 : UINT_0_32;
	END_STRUCT
END_TYPE

// DUTs/ST_GetSet_E_StepSizeAdaptation
{attribute 'TcIecLibraryType'}
{attribute 'hide'}
TYPE ST_GetSet_E_StepSizeAdaptation : 
	STRUCT
		{attribute 'GUID' := '18071995-0000-0000-0000-000000000018'}
		pInst : PVOID;
		eParam : E_StepSizeAdaptation;
		 {attribute 'hide'}
		_reserved1 : UINT_0_32;
	END_STRUCT
END_TYPE

// DUTs/ST_GetSet_E_ExecutionSequence1
{attribute 'TcIecLibraryType'}
{attribute 'hide'}
TYPE ST_GetSet_E_ExecutionSequence1 : 
	STRUCT
		{attribute 'GUID' := '18071995-0000-0000-0000-000000000018'}
		pInst : PVOID;
		eParam : E_ExecutionSequence1;
		 {attribute 'hide'}
		_reserved1 : UINT_0_32;
	END_STRUCT
END_TYPE

// DUTs/ST_GetSet_E_FpExcptCtrlSet
{attribute 'TcIecLibraryType'}
{attribute 'hide'}
TYPE ST_GetSet_E_FpExcptCtrlSet : 
	STRUCT
		{attribute 'GUID' := '18071995-0000-0000-0000-000000000018'}
		pInst : PVOID;
		eParam : E_FpExcptCtrlSet;
		 {attribute 'hide'}
		_reserved1 : UINT_24_56;
	END_STRUCT
END_TYPE

// DUTs/ST_ModuleBuildInfo
(* Generated from type 'TcMgSdk.ModuleBuildInfo' *)
{attribute 'TcIecLibraryType'}
TYPE ST_ModuleBuildInfo : 
	STRUCT
		(* Generated from item 'TcBuild' *)
		nTcBuild : UDINT;
		(* Generated from item 'TcRevision' *)
		nTcRevision : UDINT;
		(* Generated from item 'Debug' *)
		bDebug : BOOL;
		 {attribute 'hide'}
		_reserved1 : ARRAY [1..3] OF USINT;
	END_STRUCT
END_TYPE

// DUTs/ST_GetSet_ST_ModuleBuildInfo
{attribute 'TcIecLibraryType'}
{attribute 'hide'}
TYPE ST_GetSet_ST_ModuleBuildInfo : 
	STRUCT
		{attribute 'GUID' := '18071995-0000-0000-0000-000000000018'}
		pInst : PVOID;
		stParam : ST_ModuleBuildInfo;
		 {attribute 'hide'}
		_reserved1 : UINT_0_32;
	END_STRUCT
END_TYPE

// DUTs/ST_LibraryInfo
(* Generated from type 'TcMgSdk.LibraryInfo' *)
{attribute 'TcIecLibraryType'}
TYPE ST_LibraryInfo : 
	STRUCT
		(* Generated from item 'FileVersion' *)
		nFileVersion : ARRAY [0..3] OF UDINT;
		(* Generated from item 'ProductVersion' *)
		nProductVersion : ARRAY [0..3] OF UDINT;
		(* Generated from item 'VendorName' *)
		{attribute 'GUID' := '18071995-0000-0000-0000-00010000007F'}
		sVendorName : STRING(127);
		(* Generated from item 'LibraryName' *)
		{attribute 'GUID' := '18071995-0000-0000-0000-00010000007F'}
		sLibraryName : STRING(127);
		(* Generated from item 'LibraryVersion' *)
		nLibraryVersion : ARRAY [0..3] OF UDINT;
		(* Generated from item 'LibraryId' *)
		{attribute 'GUID' := '18071995-0000-0000-0000-00010000007F'}
		sLibraryId : STRING(127);
		(* Generated from item 'LibraryGUID' *)
		{attribute 'GUID' := '18071995-0000-0000-0000-000000000024'}
		nLibraryGUID : CLSID;
		(* Generated from item 'TcSdkVersion' *)
		nTcSdkVersion : ARRAY [0..3] OF UDINT;
		(* Generated from item 'Compiler' *)
		{attribute 'GUID' := '18071995-0000-0000-0000-00010000007F'}
		sCompiler : STRING(127);
		(* Generated from item 'Debug' *)
		bDebug : BOOL;
		 {attribute 'hide'}
		_reserved1 : ARRAY [1..7] OF USINT;
	END_STRUCT
END_TYPE

// DUTs/ST_GetSet_ST_LibraryInfo
{attribute 'TcIecLibraryType'}
{attribute 'hide'}
TYPE ST_GetSet_ST_LibraryInfo : 
	STRUCT
		{attribute 'GUID' := '18071995-0000-0000-0000-000000000018'}
		pInst : PVOID;
		stParam : ST_LibraryInfo;
	END_STRUCT
END_TYPE

// DUTs/ST_ModuleInfo
(* Generated from type 'TcMgSdk.ModuleInfo' *)
{attribute 'TcIecLibraryType'}
TYPE ST_ModuleInfo : 
	STRUCT
		(* Generated from item 'ClassName' *)
		{attribute 'GUID' := '18071995-0000-0000-0000-00010000007F'}
		sClassName : STRING(127);
		(* Generated from item 'CommonClassId' *)
		{attribute 'GUID' := '18071995-0000-0000-0000-000000000024'}
		nCommonClassId : CLSID;
		(* Generated from item 'VersionClassId' *)
		{attribute 'GUID' := '18071995-0000-0000-0000-000000000024'}
		nVersionClassId : CLSID;
	END_STRUCT
END_TYPE

// DUTs/ST_GetSet_ST_ModuleInfo
{attribute 'TcIecLibraryType'}
{attribute 'hide'}
TYPE ST_GetSet_ST_ModuleInfo : 
	STRUCT
		{attribute 'GUID' := '18071995-0000-0000-0000-000000000018'}
		pInst : PVOID;
		stParam : ST_ModuleInfo;
	END_STRUCT
END_TYPE

// DUTs/ST_GetSet_ST_TcMatSim_ModuleGeneratorInfo
{attribute 'TcIecLibraryType'}
{attribute 'hide'}
TYPE ST_GetSet_ST_TcMatSim_ModuleGeneratorInfo : 
	STRUCT
		{attribute 'GUID' := '18071995-0000-0000-0000-000000000018'}
		pInst : PVOID;
		stParam : ST_TcMatSim_ModuleGeneratorInfo;
	END_STRUCT
END_TYPE

// DUTs/ST_GetSet_ST_TcMatSim_SimulinkModelInfo
{attribute 'TcIecLibraryType'}
{attribute 'hide'}
TYPE ST_GetSet_ST_TcMatSim_SimulinkModelInfo : 
	STRUCT
		{attribute 'GUID' := '18071995-0000-0000-0000-000000000018'}
		pInst : PVOID;
		stParam : ST_TcMatSim_SimulinkModelInfo;
	END_STRUCT
END_TYPE

// DUTs/ST_GetSet_E_ParameterSharingType
{attribute 'TcIecLibraryType'}
{attribute 'hide'}
TYPE ST_GetSet_E_ParameterSharingType : 
	STRUCT
		{attribute 'GUID' := '18071995-0000-0000-0000-000000000018'}
		pInst : PVOID;
		eParam : E_ParameterSharingType;
		 {attribute 'hide'}
		_reserved1 : UINT_0_32;
	END_STRUCT
END_TYPE

// DUTs/ST_GetSet_ST_P_lateral_levitation_control_new_T
{attribute 'TcIecLibraryType'}
{attribute 'hide'}
TYPE ST_GetSet_ST_P_lateral_levitation_control_new_T : 
	STRUCT
		{attribute 'GUID' := '18071995-0000-0000-0000-000000000018'}
		pInst : PVOID;
		stParam : ST_P_lateral_levitation_control_new_T;
	END_STRUCT
END_TYPE

// DUTs/ST_GetSet_LREAL
{attribute 'TcIecLibraryType'}
{attribute 'hide'}
TYPE ST_GetSet_LREAL : 
	STRUCT
		{attribute 'GUID' := '18071995-0000-0000-0000-000000000018'}
		pInst : PVOID;
		fParam : LREAL;
	END_STRUCT
END_TYPE

// Version/Global_Version
{attribute 'TcGenerated'}
// This function has been automatically generated from the project information.
VAR_GLOBAL CONSTANT
	{attribute 'const_non_replaced'}
	{attribute 'linkalways'}
	stLibVersion_lateral_levitation_control_new : ST_LibVersion := (iMajor := 0, iMinor := 0, iBuild := 0, iRevision := 4, nFlags := 0, sVersion := '0.0.0.4');
	{attribute 'const_non_replaced'}
	{attribute 'linkalways'}
	sLibraryId_lateral_levitation_control_new : String := 'TE140x Module Vendor|lateral_levitation_control_new|0.0.0.4';
END_VAR

// POUs/FB_lateral_levitation_control_new

{attribute 'c++_compatible'}
{attribute 'external_name' := 'FB_lateral_levitation_control_new_GUID_BB7FAFFF_7202_35F5_7542_EB784248C869'}
{attribute 'TcIecLibraryType'}
{attribute 'reflection'}
FUNCTION_BLOCK FB_lateral_levitation_control_new
VAR
	{attribute 'hide'}
	{attribute 'no_copy'}
	{attribute 'GUID' := '18071995-0000-0000-0000-000000000018'}
	m_pData : PVOID;
	{attribute 'TcInitSymbol'}
	{attribute 'GUID' := '8007AE3B-86BB-40F2-B385-EF87FCC239A4'}
	eTraceLevelMax : TcTraceLevel := TcTraceLevel.tlInfo;
	 {attribute 'hide'}
	_reserved1 : UDINT;
	{attribute 'hide'}
	{attribute 'instance-path'}
	{attribute 'noinit'}
	{attribute 'GUID' := '18071995-0000-0000-0000-0001000000FF'}
	sInstancePath : STRING(255);
	{attribute 'hide'}
	{attribute 'noinit'}
	{attribute 'GUID' := '18071995-0000-0000-0000-000000000019'}
	m_HResultLog : HRESULT;
	{attribute 'hide'}
	{attribute 'noinit'}
	{attribute 'GUID' := '18071995-0000-0000-0000-000000000019'}
	m_HResult : HRESULT;
	 {attribute 'hide'}
	_reserved2 : ARRAY [1..184] OF USINT;
	{attribute 'hide'}
	{attribute 'no_copy'}
	m_ExtModeData : ULINT;
END_VAR
VAR_INPUT
	(* Generated from item 'y' *)
	fy : LREAL;
	(* Generated from item 'yaw' *)
	fyaw : LREAL;
	(* Generated from item 'motor_Fx_l' *)
	fmotor_Fx_l : LREAL;
	(* Generated from item 'motor_Fx_r' *)
	fmotor_Fx_r : LREAL;
	(* Generated from item 'motor_Fy_l' *)
	fmotor_Fy_l : LREAL;
	(* Generated from item 'motor_Fy_r' *)
	fmotor_Fy_r : LREAL;
	(* Generated from item 'z' *)
	fz : LREAL;
END_VAR
VAR_OUTPUT
	(* Generated from item 'F_latreq' *)
	aF_latreq : T_matrix2xdouble;
	(* Generated from item 'I_ems' *)
	aI_ems : T_matrix4xdouble;
	(* Generated from item 'F_emsfb' *)
	aF_emsfb : T_matrix2xdouble;
	(* Generated from item 'airgaps' *)
	aairgaps : T_matrix4xdouble;
	(* Generated from item 'integrals' *)
	aintegrals : T_matrix2xdouble;
	(* Generated from item 't_peak' *)
	at_peak : T_matrix2xdouble;
	(* Generated from item 'tau_x_ems' *)
	ftau_x_ems : LREAL;
END_VAR
VAR
	{attribute 'no_copy'}
	Plateral_levitation_control_new_M : POINTER TO ST_RT_MODEL_lateral_levitation_control_new_T;
END_VAR

{attribute 'TcTypeSystem'}

METHOD FB_exit : BOOL
VAR_INPUT
	bInCopyCode : BOOL;
END_VAR
END_METHOD

{attribute 'TcTypeSystem'}

METHOD FB_init : BOOL
VAR_INPUT
	bInitRetains : BOOL;
	bInCopyCode : BOOL;
END_VAR
END_METHOD

{attribute 'TcTypeSystem'}

{attribute 'monitoring' := 'call'}
	PROPERTY nHResult : HRESULT
GET
END_GET
END_PROPERTY

{attribute 'TcTypeSystem'}

{attribute 'monitoring' := 'call'}
	PROPERTY eInitExceptionHandling : E_FpExcptCtrlSetEx
GET
END_GET
SET
END_SET
END_PROPERTY

{attribute 'TcTypeSystem'}

{attribute 'monitoring' := 'call'}
	PROPERTY eUpdateExceptionHandling : E_FpExcptCtrlSetEx
GET
END_GET
SET
END_SET
END_PROPERTY

{attribute 'TcTypeSystem'}

{attribute 'monitoring' := 'call'}
	PROPERTY nExceptionCnt : ULINT
GET
END_GET
END_PROPERTY

{attribute 'TcTypeSystem'}

{attribute 'monitoring' := 'variable'}
	PROPERTY stActiveException : ST_ExceptionInfo
GET
END_GET
END_PROPERTY

{attribute 'TcTypeSystem'}

{attribute 'monitoring' := 'call'}
	PROPERTY bInitialized : BOOL
GET
END_GET
END_PROPERTY

{attribute 'TcTypeSystem'}

{attribute 'monitoring' := 'call'}
	PROPERTY bExecute : BOOL
GET
END_GET
SET
END_SET
END_PROPERTY

END_FUNCTION_BLOCK

// POUs/TcCOM Wrapper/FB_lateral_levitation_control_new_TcCOM_InitStruct

{attribute 'c++_compatible'}
{attribute 'external_name' := 'FB_lateral_levitation_control_new_TcCOM_InitStruct_GUID_97F50AE9_0319_CA3E_50BC_CCBB27B63FE3'}
{attribute 'TcIecLibraryType'}
{attribute 'call_after_init'}
{attribute 'reflection'}
FUNCTION_BLOCK FB_lateral_levitation_control_new_TcCOM_InitStruct
VAR
	{attribute 'hide'}
	{attribute 'no_copy'}
	{attribute 'GUID' := '18071995-0000-0000-0000-000000000018'}
	m_pData : PVOID;
	{attribute 'TcInitSymbol'}
	{attribute 'GUID' := '8007AE3B-86BB-40F2-B385-EF87FCC239A4'}
	eTraceLevelMaxFB : TcTraceLevel := TcTraceLevel.tlInfo;
	 {attribute 'hide'}
	_reserved1 : UDINT;
	{attribute 'hide'}
	{attribute 'instance-path'}
	{attribute 'noinit'}
	{attribute 'GUID' := '18071995-0000-0000-0000-0001000000FF'}
	sInstancePath : STRING(255);
	{attribute 'hide'}
	{attribute 'noinit'}
	{attribute 'GUID' := '18071995-0000-0000-0000-000000000019'}
	m_HResultLog : HRESULT;
	{attribute 'hide'}
	{attribute 'noinit'}
	{attribute 'GUID' := '18071995-0000-0000-0000-000000000019'}
	m_HResult : HRESULT;
	 {attribute 'hide'}
	_reserved2 : UINT_0_32;
	 {attribute 'hide'}
	_reserved3 : ARRAY [1..12] OF UINT_8_16;
	 {attribute 'hide'}
	_reserved4 : ARRAY [1..12] OF USINT;
END_VAR
VAR_INPUT
	stlateral_levitation_control_new_U : ST_lateral_levitation_control_new_U_T;
END_VAR
VAR_OUTPUT
	stlateral_levitation_control_new_Y : ST_lateral_levitation_control_new_Y_T;
END_VAR
VAR
	{attribute 'hide'}
	{attribute 'GUID' := '80FAA5A7-0B62-AEE3-90DE-6C92E3F0BFBE'}
	_iplateral_levitation_control_new : POINTER TO ITclateral_levitation_control_new;
	stInit : ST_FB_lateral_levitation_control_new_TcCOM_InitStruct;
END_VAR

{attribute 'TcTypeSystem'}

METHOD FB_init : BOOL
VAR_INPUT
	bInitRetains : BOOL;
	bInCopyCode : BOOL;
	{attribute 'GUID' := '9BDDDED0-9E85-8834-BB50-577DDDD85E40'}
	stInit : REFERENCE TO ST_FB_lateral_levitation_control_new_TcCOM_InitStruct;
END_VAR
END_METHOD

{attribute 'TcTypeSystem'}

{attribute 'call_after_init'}
METHOD FB_afterinit : BOOL
END_METHOD

{attribute 'TcTypeSystem'}

METHOD Reinit : BOOL
VAR_INPUT
	{attribute 'GUID' := '9BDDDED0-9E85-8834-BB50-577DDDD85E40'}
	stReInit : ST_FB_lateral_levitation_control_new_TcCOM_InitStruct;
END_VAR
END_METHOD

{attribute 'TcTypeSystem'}

METHOD FB_exit : BOOL
VAR_INPUT
	bInCopyCode : BOOL;
END_VAR
END_METHOD

{attribute 'TcTypeSystem'}

	PROPERTY eObjectState : TCOM_STATE
GET
END_GET
SET
END_SET
END_PROPERTY

{attribute 'TcTypeSystem'}

{attribute 'monitoring' := 'call'}
	PROPERTY nHResult : HRESULT
GET
END_GET
END_PROPERTY

{attribute 'TcTypeSystem'}

	PROPERTY ipTcComObject : ITComObject
GET
END_GET
END_PROPERTY

{attribute 'TcTypeSystem'}

	PROPERTY ipADI : ITcADI
GET
END_GET
END_PROPERTY

{attribute 'TcTypeSystem'}

{attribute 'monitoring' := 'call'}
	PROPERTY nTaskOid : OTCID
GET
END_GET
SET
END_SET
END_PROPERTY

{attribute 'TcTypeSystem'}

{attribute 'monitoring' := 'call'}
	PROPERTY nTaskPriority : UDINT
GET
END_GET
END_PROPERTY

{attribute 'TcTypeSystem'}

{attribute 'monitoring' := 'call'}
	PROPERTY nTaskCycleTimeNs : UDINT
GET
END_GET
END_PROPERTY

{attribute 'TcTypeSystem'}

{attribute 'monitoring' := 'call'}
	PROPERTY nTaskPort : UINT
GET
END_GET
END_PROPERTY

{attribute 'TcTypeSystem'}

{attribute 'monitoring' := 'call'}
	PROPERTY nTaskSortOrder : UDINT
GET
END_GET
SET
END_SET
END_PROPERTY

{attribute 'TcTypeSystem'}

{attribute 'monitoring' := 'call'}
	PROPERTY eTraceLevelMax : TcTraceLevel
GET
END_GET
SET
END_SET
END_PROPERTY

{attribute 'TcTypeSystem'}

{attribute 'monitoring' := 'call'}
	PROPERTY eModuleCaller : E_ModuleCaller
GET
END_GET
SET
END_SET
END_PROPERTY

{attribute 'TcTypeSystem'}

{attribute 'monitoring' := 'call'}
	PROPERTY eCallerVerification : E_CallerVerification
GET
END_GET
SET
END_SET
END_PROPERTY

{attribute 'TcTypeSystem'}

{attribute 'monitoring' := 'call'}
	PROPERTY eStepSizeAdaptation : E_StepSizeAdaptation
GET
END_GET
SET
END_SET
END_PROPERTY

{attribute 'TcTypeSystem'}

{attribute 'monitoring' := 'call'}
	PROPERTY eExecutionSequence : E_ExecutionSequence1
GET
END_GET
SET
END_SET
END_PROPERTY

{attribute 'TcTypeSystem'}

{attribute 'monitoring' := 'call'}
	PROPERTY bExecute : BOOL
GET
END_GET
SET
END_SET
END_PROPERTY

{attribute 'TcTypeSystem'}

{attribute 'monitoring' := 'call'}
	PROPERTY eAccessLockState : TCOM_STATE
GET
END_GET
SET
END_SET
END_PROPERTY

{attribute 'TcTypeSystem'}

{attribute 'monitoring' := 'call'}
	PROPERTY eInitExceptionHandling : E_FpExcptCtrlSet
GET
END_GET
SET
END_SET
END_PROPERTY

{attribute 'TcTypeSystem'}

{attribute 'monitoring' := 'call'}
	PROPERTY eUpdateExceptionHandling : E_FpExcptCtrlSetEx
GET
END_GET
SET
END_SET
END_PROPERTY

{attribute 'TcTypeSystem'}

{attribute 'monitoring' := 'variable'}
	PROPERTY stModuleBuildInfo : ST_ModuleBuildInfo
GET
END_GET
END_PROPERTY

{attribute 'TcTypeSystem'}

{attribute 'monitoring' := 'call'}
	PROPERTY bInitialized : BOOL
GET
END_GET
END_PROPERTY

{attribute 'TcTypeSystem'}

{attribute 'monitoring' := 'call'}
	PROPERTY nSkippedExecutionCount : UDINT
GET
END_GET
END_PROPERTY

{attribute 'TcTypeSystem'}

{attribute 'monitoring' := 'variable'}
	PROPERTY stLibraryInfo : ST_LibraryInfo
GET
END_GET
END_PROPERTY

{attribute 'TcTypeSystem'}

{attribute 'monitoring' := 'variable'}
	PROPERTY stModuleInfo : ST_ModuleInfo
GET
END_GET
END_PROPERTY

{attribute 'TcTypeSystem'}

{attribute 'monitoring' := 'variable'}
	PROPERTY stModuleGeneratorInfo : ST_TcMatSim_ModuleGeneratorInfo
GET
END_GET
SET
END_SET
END_PROPERTY

{attribute 'TcTypeSystem'}

{attribute 'monitoring' := 'variable'}
	PROPERTY stSimulinkModelInfo : ST_TcMatSim_SimulinkModelInfo
GET
END_GET
SET
END_SET
END_PROPERTY

{attribute 'TcTypeSystem'}

{attribute 'monitoring' := 'call'}
	PROPERTY elateral_levitation_control_new_P_Sharing : E_ParameterSharingType
GET
END_GET
SET
END_SET
END_PROPERTY

{attribute 'TcTypeSystem'}

{attribute 'monitoring' := 'call'}
	PROPERTY nlateral_levitation_control_new_P_Definer : OTCID
GET
END_GET
END_PROPERTY

{attribute 'TcTypeSystem'}

{attribute 'monitoring' := 'variable'}
	PROPERTY stlateral_levitation_control_new_P : ST_P_lateral_levitation_control_new_T
GET
END_GET
SET
END_SET
END_PROPERTY

{attribute 'TcTypeSystem'}

{attribute 'monitoring' := 'call'}
	PROPERTY fSimulationTime : LREAL
GET
END_GET
END_PROPERTY

{attribute 'TcTypeSystem'}

{attribute 'monitoring' := 'call'}
	PROPERTY nCycleCount : ULINT
GET
END_GET
END_PROPERTY

{attribute 'TcTypeSystem'}

{attribute 'monitoring' := 'call'}
	PROPERTY nExceptionCount : ULINT
GET
END_GET
END_PROPERTY

{attribute 'TcTypeSystem'}

{attribute 'monitoring' := 'variable'}
	PROPERTY stExceptionInfo : ST_ExceptionInfo
GET
END_GET
END_PROPERTY

END_FUNCTION_BLOCK
